LIN {X 0,Y 523.977,Z 285.218,A -85,B 0,C 180,E1 -4797.718,E2 -4797.718} C_VEL
LIN {X 0,Y 523.948,Z 285.216,A -85,B 0,C 180,E1 -4800.855,E2 -4800.855} C_VEL
LIN {X 0,Y 523.962,Z 285.215,A -85,B 0,C 180,E1 -4803.734,E2 -4803.734} C_VEL
LIN {X 0,Y 523.905,Z 285.226,A -85,B 0,C 180,E1 -4806.401,E2 -4806.401} C_VEL
LIN {X 0,Y 523.921,Z 285.217,A -85,B 0,C 180,E1 -4809.085,E2 -4809.085} C_VEL
LIN {X 0,Y 523.954,Z 285.219,A -85,B 0,C 180,E1 -4812.119,E2 -4812.119} C_VEL
LIN {X 0,Y 523.941,Z 285.215,A -85,B 0,C 180,E1 -4815.31,E2 -4815.31} C_VEL
LIN {X 0,Y 523.959,Z 285.219,A -85,B 0,C 180,E1 -4818.689,E2 -4818.689} C_VEL
LIN {X 0,Y 523.912,Z 285.219,A -85,B 0,C 180,E1 -4821.898,E2 -4821.898} C_VEL
LIN {X 0,Y 523.93,Z 285.222,A -85,B 0,C 180,E1 -4824.909,E2 -4824.909} C_VEL
LIN {X 0,Y 523.937,Z 285.215,A -85,B 0,C 180,E1 -4827.678,E2 -4827.678} C_VEL
LIN {X 0,Y 523.956,Z 285.221,A -85,B 0,C 180,E1 -4830.674,E2 -4830.674} C_VEL
LIN {X 0,Y 523.97,Z 285.211,A -85,B 0,C 180,E1 -4833.728,E2 -4833.728} C_VEL
LIN {X 0,Y 523.928,Z 285.217,A -85,B 0,C 180,E1 -4836.27,E2 -4836.27} C_VEL
LIN {X 0,Y 523.936,Z 285.222,A -85,B 0,C 180,E1 -4838.766,E2 -4838.766} C_VEL
LIN {X 0,Y 523.941,Z 285.222,A -85,B 0,C 180,E1 -4841.22,E2 -4841.22} C_VEL
LIN {X 0,Y 523.924,Z 285.219,A -85,B 0,C 180,E1 -4843.638,E2 -4843.638} C_VEL
LIN {X 0,Y 523.927,Z 285.216,A -85,B 0,C 180,E1 -4846.028,E2 -4846.028} C_VEL
LIN {X 0,Y 524.002,Z 285.207,A -85,B 0,C 180,E1 -4848.394,E2 -4848.394} C_VEL
LIN {X 0,Y 523.991,Z 285.215,A -85,B 0,C 180,E1 -4851.516,E2 -4851.516} C_VEL
LIN {X 0,Y 524.07,Z 285.199,A -85,B 0,C 180,E1 -4854.614,E2 -4854.614} C_VEL
LIN {X 0,Y 524.095,Z 285.201,A -85,B 0,C 180,E1 -4857.694,E2 -4857.694} C_VEL
LIN {X 0,Y 524.109,Z 285.194,A -85,B 0,C 180,E1 -4860.768,E2 -4860.768} C_VEL
LIN {X 0,Y 524.058,Z 285.203,A -85,B 0,C 180,E1 -4863.075,E2 -4863.075} C_VEL
LIN {X 0,Y 524.011,Z 285.208,A -85,B 0,C 180,E1 -4866.159,E2 -4866.159} C_VEL
LIN {X 0,Y 523.979,Z 285.213,A -85,B 0,C 180,E1 -4869.262,E2 -4869.262} C_VEL
LIN {X 0,Y 523.986,Z 285.219,A -85,B 0,C 180,E1 -4871.737,E2 -4871.737} C_VEL
LIN {X 0,Y 523.979,Z 285.21,A -85,B 0,C 180,E1 -4875.051,E2 -4875.051} C_VEL
LIN {X 0,Y 523.934,Z 285.225,A -85,B 0,C 180,E1 -4877.97,E2 -4877.97} C_VEL
LIN {X 0,Y 523.94,Z 285.218,A -85,B 0,C 180,E1 -4880.411,E2 -4880.411} C_VEL
LIN {X 0,Y 523.897,Z 285.22,A -85,B 0,C 180,E1 -4882.894,E2 -4882.894} C_VEL
LIN {X 0,Y 523.89,Z 285.222,A -85,B 0,C 180,E1 -4885.422,E2 -4885.422} C_VEL
LIN {X 0,Y 523.888,Z 285.229,A -85,B 0,C 180,E1 -4888.004,E2 -4888.004} C_VEL
LIN {X 0,Y 523.927,Z 285.218,A -85,B 0,C 180,E1 -4890.853,E2 -4890.853} C_VEL
LIN {X 0,Y 523.919,Z 285.219,A -85,B 0,C 180,E1 -4893.729,E2 -4893.729} C_VEL
LIN {X 0,Y 523.853,Z 285.235,A -85,B 0,C 180,E1 -4896.395,E2 -4896.395} C_VEL
LIN {X 0,Y 523.89,Z 285.222,A -85,B 0,C 180,E1 -4899.088,E2 -4899.088} C_VEL
LIN {X 0,Y 523.881,Z 285.226,A -85,B 0,C 180,E1 -4902.126,E2 -4902.126} C_VEL
LIN {X 0,Y 523.927,Z 285.217,A -85,B 0,C 180,E1 -4905.312,E2 -4905.312} C_VEL
LIN {X 0,Y 523.865,Z 285.229,A -85,B 0,C 180,E1 -4906.891,E2 -4906.891} C_VEL
LIN {X 0,Y 523.18,Z 285.312,A -85,B 0,C 180,E1 -4907.532,E2 -4907.532} C_VEL
LIN {X 0,Y 520.318,Z 285.675,A -85,B 0,C 180,E1 -4908.574,E2 -4908.574} C_VEL
LIN {X 0,Y 517.917,Z 285.971,A -85,B 0,C 180,E1 -4909.412,E2 -4909.412} C_VEL
LIN {X 0,Y 516.897,Z 286.095,A -85,B 0,C 180,E1 -4910.06,E2 -4910.06} C_VEL
LIN {X 0,Y 516.819,Z 286.105,A -85,B 0,C 180,E1 -4910.279,E2 -4910.279} C_VEL
LIN {X 0,Y 516.79,Z 286.108,A -85,B 0,C 180,E1 -4913.247,E2 -4913.247} C_VEL
LIN {X 0,Y 516.836,Z 286.101,A -85,B 0,C 180,E1 -4916.115,E2 -4916.115} C_VEL
LIN {X 0,Y 516.85,Z 286.107,A -85,B 0,C 180,E1 -4918.944,E2 -4918.944} C_VEL
LIN {X 0,Y 516.858,Z 286.097,A -85,B 0,C 180,E1 -4922.11,E2 -4922.11} C_VEL
LIN {X 0,Y 516.829,Z 286.11,A -85,B 0,C 180,E1 -4925.067,E2 -4925.067} C_VEL
LIN {X 0,Y 516.875,Z 286.097,A -85,B 0,C 180,E1 -4927.621,E2 -4927.621} C_VEL
LIN {X 0,Y 516.92,Z 286.089,A -85,B 0,C 180,E1 -4930.128,E2 -4930.128} C_VEL
LIN {X 0,Y 516.879,Z 286.101,A -85,B 0,C 180,E1 -4933.408,E2 -4933.408} C_VEL
LIN {X 0,Y 516.879,Z 286.096,A -85,B 0,C 180,E1 -4935.832,E2 -4935.832} C_VEL
LIN {X 0,Y 516.946,Z 286.09,A -85,B 0,C 180,E1 -4939.026,E2 -4939.026} C_VEL
LIN {X 0,Y 516.926,Z 286.089,A -85,B 0,C 180,E1 -4942.184,E2 -4942.184} C_VEL
LIN {X 0,Y 516.988,Z 286.081,A -85,B 0,C 180,E1 -4944.537,E2 -4944.537} C_VEL
LIN {X 0,Y 517.076,Z 286.078,A -85,B 0,C 180,E1 -4947.661,E2 -4947.661} C_VEL
LIN {X 0,Y 517.068,Z 286.075,A -85,B 0,C 180,E1 -4949.997,E2 -4949.997} C_VEL
LIN {X 0,Y 517.076,Z 286.071,A -85,B 0,C 180,E1 -4952.334,E2 -4952.334} C_VEL
LIN {X 0,Y 516.975,Z 286.087,A -85,B 0,C 180,E1 -4956.241,E2 -4956.241} C_VEL
LIN {X 0,Y 516.935,Z 286.093,A -85,B 0,C 180,E1 -4959.386,E2 -4959.386} C_VEL
LIN {X 0,Y 516.964,Z 286.096,A -85,B 0,C 180,E1 -4962.161,E2 -4962.161} C_VEL
LIN {X 0,Y 517.499,Z 292.038,A -85,B 0,C 180,E1 -4963.345,E2 -4963.345} C_VEL
LIN {X 0,Y 517.273,Z 306.74,A -85,B 0,C 180,E1 -4966.168,E2 -4966.168} C_VEL
LIN {X 0,Y 517.259,Z 309.78,A -85,B 0,C 180,E1 -4966.701,E2 -4966.701} C_VEL
LIN {X 0,Y 519.063,Z 319.454,A -85,B 0,C 180,E1 -4966.895,E2 -4966.895} C_VEL
LIN {X 0,Y 518.594,Z 416.572,A -85,B 0,C 180,E1 -4968.272,E2 -4968.272} C_VEL
LIN {X 0,Y 518.456,Z 429.396,A -85,B 0,C 180,E1 -4968.609,E2 -4968.609} C_VEL
LIN {X 0,Y 518.201,Z 441.954,A -85,B 0,C 180,E1 -4969.094,E2 -4969.094} C_VEL
LIN {X 0,Y 517.926,Z 453.888,A -85,B 0,C 180,E1 -4969.723,E2 -4969.723} C_VEL
LIN {X 0,Y 517.565,Z 465.513,A -85,B 0,C 180,E1 -4970.517,E2 -4970.517} C_VEL
LIN {X 0,Y 517.293,Z 475.939,A -85,B 0,C 180,E1 -4971.411,E2 -4971.411} C_VEL
LIN {X 0,Y 517.017,Z 485.499,A -85,B 0,C 180,E1 -4972.429,E2 -4972.429} C_VEL
LIN {X 0,Y 516.759,Z 494.699,A -85,B 0,C 180,E1 -4973.649,E2 -4973.649} C_VEL
LIN {X 0,Y 516.619,Z 500.444,A -85,B 0,C 180,E1 -4974.582,E2 -4974.582} C_VEL
LIN {X 0,Y 516.472,Z 506.637,A -85,B 0,C 180,E1 -4975.809,E2 -4975.809} C_VEL
LIN {X 0,Y 516.367,Z 511.787,A -85,B 0,C 180,E1 -4977.121,E2 -4977.121} C_VEL
LIN {X 0,Y 516.249,Z 515.595,A -85,B 0,C 180,E1 -4978.45,E2 -4978.45} C_VEL
LIN {X 0,Y 516.228,Z 517.529,A -85,B 0,C 180,E1 -4979.389,E2 -4979.389} C_VEL
LIN {X 0,Y 516.199,Z 518.78,A -85,B 0,C 180,E1 -4980.243,E2 -4980.243} C_VEL
LIN {X 0,Y 516.173,Z 519.558,A -85,B 0,C 180,E1 -4981.152,E2 -4981.152} C_VEL
LIN {X 0,Y 516.192,Z 519.773,A -85,B 0,C 180,E1 -4982.42,E2 -4982.42} C_VEL
LIN {X 0,Y 516.205,Z 518.701,A -85,B 0,C 180,E1 -4983.926,E2 -4983.926} C_VEL
LIN {X 0,Y 516.201,Z 516.554,A -85,B 0,C 180,E1 -4985.225,E2 -4985.225} C_VEL
LIN {X 0,Y 516.327,Z 513.062,A -85,B 0,C 180,E1 -4986.574,E2 -4986.574} C_VEL
LIN {X 0,Y 516.434,Z 508.387,A -85,B 0,C 180,E1 -4987.879,E2 -4987.879} C_VEL
LIN {X 0,Y 516.566,Z 502.458,A -85,B 0,C 180,E1 -4989.149,E2 -4989.149} C_VEL
LIN {X 0,Y 516.787,Z 495.044,A -85,B 0,C 180,E1 -4990.397,E2 -4990.397} C_VEL
LIN {X 0,Y 517.023,Z 485.936,A -85,B 0,C 180,E1 -4991.614,E2 -4991.614} C_VEL
LIN {X 0,Y 517.316,Z 476.332,A -85,B 0,C 180,E1 -4992.648,E2 -4992.648} C_VEL
LIN {X 0,Y 517.581,Z 466.186,A -85,B 0,C 180,E1 -4993.526,E2 -4993.526} C_VEL
LIN {X 0,Y 517.857,Z 455.616,A -85,B 0,C 180,E1 -4994.264,E2 -4994.264} C_VEL
LIN {X 0,Y 518.159,Z 443.921,A -85,B 0,C 180,E1 -4994.908,E2 -4994.908} C_VEL
LIN {X 0,Y 518.447,Z 431.069,A -85,B 0,C 180,E1 -4995.429,E2 -4995.429} C_VEL
LIN {X 0,Y 518.619,Z 417.781,A -85,B 0,C 180,E1 -4995.792,E2 -4995.792} C_VEL
LIN {X 0,Y 518.817,Z 379.999,A -85,B 0,C 180,E1 -4996.349,E2 -4996.349} C_VEL
LIN {X 0,Y 519.087,Z 319.542,A -85,B 0,C 180,E1 -4997.195,E2 -4997.195} C_VEL
LIN {X 0,Y 517.182,Z 309.105,A -85,B 0,C 180,E1 -4997.415,E2 -4997.415} C_VEL
LIN {X 0,Y 517.275,Z 293.741,A -85,B 0,C 180,E1 -5000.121,E2 -5000.121} C_VEL
LIN {X 0,Y 516.989,Z 286.453,A -85,B 0,C 180,E1 -5001.398,E2 -5001.398} C_VEL
LIN {X 0,Y 516.922,Z 286.097,A -85,B 0,C 180,E1 -5001.497,E2 -5001.497} C_VEL
LIN {X 0,Y 516.844,Z 286.105,A -85,B 0,C 180,E1 -5004.664,E2 -5004.664} C_VEL
LIN {X 0,Y 516.858,Z 286.099,A -85,B 0,C 180,E1 -5007.452,E2 -5007.452} C_VEL
LIN {X 0,Y 516.89,Z 286.099,A -85,B 0,C 180,E1 -5010.693,E2 -5010.693} C_VEL
LIN {X 0,Y 516.9,Z 286.097,A -85,B 0,C 180,E1 -5013.8,E2 -5013.8} C_VEL
LIN {X 0,Y 516.823,Z 286.109,A -85,B 0,C 180,E1 -5016.774,E2 -5016.774} C_VEL
LIN {X 0,Y 516.887,Z 286.096,A -85,B 0,C 180,E1 -5019.73,E2 -5019.73} C_VEL
LIN {X 0,Y 516.876,Z 286.105,A -85,B 0,C 180,E1 -5022.594,E2 -5022.594} C_VEL
LIN {X 0,Y 516.887,Z 286.098,A -85,B 0,C 180,E1 -5025.028,E2 -5025.028} C_VEL
LIN {X 0,Y 516.91,Z 286.095,A -85,B 0,C 180,E1 -5028.232,E2 -5028.232} C_VEL
LIN {X 0,Y 516.915,Z 286.091,A -85,B 0,C 180,E1 -5031.399,E2 -5031.399} C_VEL
LIN {X 0,Y 516.949,Z 286.086,A -85,B 0,C 180,E1 -5033.756,E2 -5033.756} C_VEL
LIN {X 0,Y 516.99,Z 286.089,A -85,B 0,C 180,E1 -5036.883,E2 -5036.883} C_VEL
LIN {X 0,Y 517.023,Z 286.074,A -85,B 0,C 180,E1 -5040,E2 -5040} C_VEL
LIN {X 0,Y 516.994,Z 286.085,A -85,B 0,C 180,E1 -5043.117,E2 -5043.117} C_VEL
LIN {X 0,Y 516.957,Z 286.086,A -85,B 0,C 180,E1 -5046.244,E2 -5046.244} C_VEL
LIN {X 0,Y 516.914,Z 286.095,A -85,B 0,C 180,E1 -5049.39,E2 -5049.39} C_VEL
LIN {X 0,Y 516.929,Z 286.086,A -85,B 0,C 180,E1 -5051.825,E2 -5051.825} C_VEL
LIN {X 0,Y 516.903,Z 286.099,A -85,B 0,C 180,E1 -5055.153,E2 -5055.153} C_VEL
LIN {X 0,Y 516.878,Z 286.094,A -85,B 0,C 180,E1 -5058.224,E2 -5058.224} C_VEL
LIN {X 0,Y 516.869,Z 286.095,A -85,B 0,C 180,E1 -5060.703,E2 -5060.703} C_VEL
LIN {X 0,Y 516.866,Z 286.104,A -85,B 0,C 180,E1 -5063.224,E2 -5063.224} C_VEL
LIN {X 0,Y 516.904,Z 286.091,A -85,B 0,C 180,E1 -5066.201,E2 -5066.201} C_VEL
LIN {X 0,Y 516.898,Z 286.098,A -85,B 0,C 180,E1 -5069.306,E2 -5069.306} C_VEL
LIN {X 0,Y 516.866,Z 286.096,A -85,B 0,C 180,E1 -5072.549,E2 -5072.549} C_VEL
LIN {X 0,Y 516.851,Z 286.105,A -85,B 0,C 180,E1 -5075.337,E2 -5075.337} C_VEL
LIN {X 0,Y 516.858,Z 286.101,A -85,B 0,C 180,E1 -5077.949,E2 -5077.949} C_VEL
LIN {X 0,Y 516.887,Z 286.095,A -85,B 0,C 180,E1 -5080.741,E2 -5080.741} C_VEL
LIN {X 0,Y 516.851,Z 286.107,A -85,B 0,C 180,E1 -5083.907,E2 -5083.907} C_VEL
LIN {X 0,Y 516.852,Z 286.104,A -85,B 0,C 180,E1 -5086.111,E2 -5086.111} C_VEL
LIN {X 0,Y 516.889,Z 286.098,A -85,B 0,C 180,E1 -5089.266,E2 -5089.266} C_VEL
LIN {X 0,Y 516.862,Z 286.104,A -85,B 0,C 180,E1 -5092.06,E2 -5092.06} C_VEL
LIN {X 0,Y 516.875,Z 286.098,A -85,B 0,C 180,E1 -5095.18,E2 -5095.18} C_VEL
LIN {X 0,Y 516.865,Z 286.107,A -85,B 0,C 180,E1 -5097.98,E2 -5097.98} C_VEL
LIN {X 0,Y 516.92,Z 286.094,A -85,B 0,C 180,E1 -5100.7,E2 -5100.7} C_VEL
LIN {X 0,Y 516.931,Z 286.097,A -85,B 0,C 180,E1 -5103.807,E2 -5103.807} C_VEL
LIN {X 0,Y 516.948,Z 286.248,A -85,B 0,C 180,E1 -5105.43,E2 -5105.43} C_VEL
LIN {X 0,Y 518.381,Z 294.852,A -85,B 0,C 180,E1 -5106.853,E2 -5106.853} C_VEL
LIN {X 0,Y 517.942,Z 314.961,A -85,B 0,C 180,E1 -5109.982,E2 -5109.982} C_VEL
LIN {X 0,Y 517.423,Z 334.741,A -85,B 0,C 180,E1 -5113.024,E2 -5113.024} C_VEL
LIN {X 0,Y 517.282,Z 345.377,A -85,B 0,C 180,E1 -5114.634,E2 -5114.634} C_VEL
LIN {X 0,Y 519.061,Z 357.7,A -85,B 0,C 180,E1 -5114.862,E2 -5114.862} C_VEL
LIN {X 0,Y 518.575,Z 454.458,A -85,B 0,C 180,E1 -5116.234,E2 -5116.234} C_VEL
LIN {X 0,Y 518.297,Z 468.259,A -85,B 0,C 180,E1 -5116.601,E2 -5116.601} C_VEL
LIN {X 0,Y 517.976,Z 481.158,A -85,B 0,C 180,E1 -5117.117,E2 -5117.117} C_VEL
LIN {X 0,Y 517.817,Z 492.708,A -85,B 0,C 180,E1 -5117.745,E2 -5117.745} C_VEL
LIN {X 0,Y 517.485,Z 504.303,A -85,B 0,C 180,E1 -5118.547,E2 -5118.547} C_VEL
LIN {X 0,Y 517.151,Z 514.547,A -85,B 0,C 180,E1 -5119.432,E2 -5119.432} C_VEL
LIN {X 0,Y 516.887,Z 523.76,A -85,B 0,C 180,E1 -5120.415,E2 -5120.415} C_VEL
LIN {X 0,Y 516.664,Z 532.738,A -85,B 0,C 180,E1 -5121.595,E2 -5121.595} C_VEL
LIN {X 0,Y 516.508,Z 539.965,A -85,B 0,C 180,E1 -5122.772,E2 -5122.772} C_VEL
LIN {X 0,Y 516.42,Z 546.546,A -85,B 0,C 180,E1 -5124.145,E2 -5124.145} C_VEL
LIN {X 0,Y 516.268,Z 550.897,A -85,B 0,C 180,E1 -5125.318,E2 -5125.318} C_VEL
LIN {X 0,Y 516.351,Z 553.206,A -85,B 0,C 180,E1 -5126.101,E2 -5126.101} C_VEL
LIN {X 0,Y 516.282,Z 555.072,A -85,B 0,C 180,E1 -5126.881,E2 -5126.881} C_VEL
LIN {X 0,Y 516.26,Z 556.472,A -85,B 0,C 180,E1 -5127.662,E2 -5127.662} C_VEL
LIN {X 0,Y 516.16,Z 558.08,A -85,B 0,C 180,E1 -5129.222,E2 -5129.222} C_VEL
LIN {X 0,Y 516.158,Z 558.297,A -85,B 0,C 180,E1 -5130.003,E2 -5130.003} C_VEL
LIN {X 0,Y 516.192,Z 557.473,A -85,B 0,C 180,E1 -5131.563,E2 -5131.563} C_VEL
LIN {X 0,Y 516.261,Z 556.479,A -85,B 0,C 180,E1 -5132.343,E2 -5132.343} C_VEL
LIN {X 0,Y 516.283,Z 555.079,A -85,B 0,C 180,E1 -5133.124,E2 -5133.124} C_VEL
LIN {X 0,Y 516.312,Z 552.136,A -85,B 0,C 180,E1 -5134.296,E2 -5134.296} C_VEL
LIN {X 0,Y 516.376,Z 548.152,A -85,B 0,C 180,E1 -5135.469,E2 -5135.469} C_VEL
LIN {X 0,Y 516.423,Z 542.925,A -85,B 0,C 180,E1 -5136.664,E2 -5136.664} C_VEL
LIN {X 0,Y 516.558,Z 536.56,A -85,B 0,C 180,E1 -5137.822,E2 -5137.822} C_VEL
LIN {X 0,Y 516.771,Z 528.505,A -85,B 0,C 180,E1 -5139,E2 -5139} C_VEL
LIN {X 0,Y 516.987,Z 520.294,A -85,B 0,C 180,E1 -5139.983,E2 -5139.983} C_VEL
LIN {X 0,Y 517.273,Z 510.282,A -85,B 0,C 180,E1 -5140.967,E2 -5140.967} C_VEL
LIN {X 0,Y 517.626,Z 500.396,A -85,B 0,C 180,E1 -5141.753,E2 -5141.753} C_VEL
LIN {X 0,Y 517.852,Z 489.209,A -85,B 0,C 180,E1 -5142.468,E2 -5142.468} C_VEL
LIN {X 0,Y 518.152,Z 476.709,A -85,B 0,C 180,E1 -5143.083,E2 -5143.083} C_VEL
LIN {X 0,Y 518.381,Z 464.379,A -85,B 0,C 180,E1 -5143.527,E2 -5143.527} C_VEL
LIN {X 0,Y 518.589,Z 451.7,A -85,B 0,C 180,E1 -5143.821,E2 -5143.821} C_VEL
LIN {X 0,Y 519.006,Z 357.028,A -85,B 0,C 180,E1 -5145.151,E2 -5145.151} C_VEL
LIN {X 0,Y 517.295,Z 345.507,A -85,B 0,C 180,E1 -5145.367,E2 -5145.367} C_VEL
LIN {X 0,Y 517.761,Z 324.652,A -85,B 0,C 180,E1 -5148.603,E2 -5148.603} C_VEL
LIN {X 0,Y 518.218,Z 306.327,A -85,B 0,C 180,E1 -5151.481,E2 -5151.481} C_VEL
LIN {X 0,Y 518.477,Z 294.562,A -85,B 0,C 180,E1 -5153.36,E2 -5153.36} C_VEL
LIN {X 0,Y 516.925,Z 286.095,A -85,B 0,C 180,E1 -5154.821,E2 -5154.821} C_VEL
LIN {X 0,Y 516.927,Z 286.095,A -85,B 0,C 180,E1 -5157.533,E2 -5157.533} C_VEL
LIN {X 0,Y 516.896,Z 286.102,A -85,B 0,C 180,E1 -5160.204,E2 -5160.204} C_VEL
LIN {X 0,Y 516.898,Z 286.092,A -85,B 0,C 180,E1 -5162.947,E2 -5162.947} C_VEL
LIN {X 0,Y 516.873,Z 286.099,A -85,B 0,C 180,E1 -5165.78,E2 -5165.78} C_VEL
LIN {X 0,Y 516.881,Z 286.097,A -85,B 0,C 180,E1 -5168.716,E2 -5168.716} C_VEL
LIN {X 0,Y 516.914,Z 286.092,A -85,B 0,C 180,E1 -5171.775,E2 -5171.775} C_VEL
LIN {X 0,Y 516.894,Z 286.094,A -85,B 0,C 180,E1 -5175.007,E2 -5175.007} C_VEL
LIN {X 0,Y 516.915,Z 286.098,A -85,B 0,C 180,E1 -5178.398,E2 -5178.398} C_VEL
LIN {X 0,Y 516.878,Z 286.095,A -85,B 0,C 180,E1 -5181.284,E2 -5181.284} C_VEL
LIN {X 0,Y 516.883,Z 286.097,A -85,B 0,C 180,E1 -5184.22,E2 -5184.22} C_VEL
LIN {X 0,Y 516.892,Z 286.097,A -85,B 0,C 180,E1 -5187.053,E2 -5187.053} C_VEL
LIN {X 0,Y 516.895,Z 286.092,A -85,B 0,C 180,E1 -5189.796,E2 -5189.796} C_VEL
LIN {X 0,Y 516.922,Z 286.093,A -85,B 0,C 180,E1 -5192.467,E2 -5192.467} C_VEL
LIN {X 0,Y 516.904,Z 286.098,A -85,B 0,C 180,E1 -5195.071,E2 -5195.071} C_VEL
LIN {X 0,Y 516.876,Z 286.097,A -85,B 0,C 180,E1 -5198.462,E2 -5198.462} C_VEL
LIN {X 0,Y 516.893,Z 286.101,A -85,B 0,C 180,E1 -5200.954,E2 -5200.954} C_VEL
LIN {X 0,Y 516.902,Z 286.096,A -85,B 0,C 180,E1 -5203.41,E2 -5203.41} C_VEL
LIN {X 0,Y 516.883,Z 286.095,A -85,B 0,C 180,E1 -5205.833,E2 -5205.833} C_VEL
LIN {X 0,Y 516.955,Z 286.085,A -85,B 0,C 180,E1 -5208.233,E2 -5208.233} C_VEL
LIN {X 0,Y 516.956,Z 286.093,A -85,B 0,C 180,E1 -5211.399,E2 -5211.399} C_VEL
LIN {X 0,Y 516.988,Z 286.084,A -85,B 0,C 180,E1 -5213.757,E2 -5213.757} C_VEL
LIN {X 0,Y 517.002,Z 286.081,A -85,B 0,C 180,E1 -5216.883,E2 -5216.883} C_VEL
LIN {X 0,Y 517.065,Z 286.074,A -85,B 0,C 180,E1 -5220,E2 -5220} C_VEL
LIN {X 0,Y 517,Z 286.082,A -85,B 0,C 180,E1 -5223.117,E2 -5223.117} C_VEL
LIN {X 0,Y 516.974,Z 286.084,A -85,B 0,C 180,E1 -5226.244,E2 -5226.244} C_VEL
LIN {X 0,Y 516.934,Z 286.092,A -85,B 0,C 180,E1 -5229.39,E2 -5229.39} C_VEL
LIN {X 0,Y 516.941,Z 286.096,A -85,B 0,C 180,E1 -5231.807,E2 -5231.807} C_VEL
LIN {X 0,Y 516.931,Z 286.089,A -85,B 0,C 180,E1 -5235.145,E2 -5235.145} C_VEL
LIN {X 0,Y 516.902,Z 286.096,A -85,B 0,C 180,E1 -5238.223,E2 -5238.223} C_VEL
LIN {X 0,Y 516.89,Z 286.094,A -85,B 0,C 180,E1 -5240.703,E2 -5240.703} C_VEL
LIN {X 0,Y 516.847,Z 286.099,A -85,B 0,C 180,E1 -5243.225,E2 -5243.225} C_VEL
LIN {X 0,Y 516.87,Z 286.104,A -85,B 0,C 180,E1 -5246.182,E2 -5246.182} C_VEL
LIN {X 0,Y 516.878,Z 286.096,A -85,B 0,C 180,E1 -5249.519,E2 -5249.519} C_VEL
LIN {X 0,Y 516.887,Z 286.099,A -85,B 0,C 180,E1 -5252.543,E2 -5252.543} C_VEL
LIN {X 0,Y 516.843,Z 286.099,A -85,B 0,C 180,E1 -5255.327,E2 -5255.327} C_VEL
LIN {X 0,Y 516.857,Z 286.102,A -85,B 0,C 180,E1 -5258.718,E2 -5258.718} C_VEL
LIN {X 0,Y 516.831,Z 286.101,A -85,B 0,C 180,E1 -5261.784,E2 -5261.784} C_VEL
LIN {X 0,Y 516.895,Z 286.095,A -85,B 0,C 180,E1 -5265.007,E2 -5265.007} C_VEL
LIN {X 0,Y 516.827,Z 286.107,A -85,B 0,C 180,E1 -5268.41,E2 -5268.41} C_VEL
LIN {X 0,Y 516.819,Z 286.105,A -85,B 0,C 180,E1 -5270.279,E2 -5270.279} C_VEL
LIN {X 0,Y 516.165,Z 286.191,A -85,B 0,C 180,E1 -5270.93,E2 -5270.93} C_VEL
LIN {X 0,Y 513.309,Z 286.543,A -85,B 0,C 180,E1 -5271.985,E2 -5271.985} C_VEL
LIN {X 0,Y 510.883,Z 286.85,A -85,B 0,C 180,E1 -5272.835,E2 -5272.835} C_VEL
LIN {X 0,Y 509.834,Z 286.973,A -85,B 0,C 180,E1 -5273.492,E2 -5273.492} C_VEL
LIN {X 0,Y 509.746,Z 286.983,A -85,B 0,C 180,E1 -5273.715,E2 -5273.715} C_VEL
LIN {X 0,Y 509.805,Z 286.98,A -85,B 0,C 180,E1 -5276.535,E2 -5276.535} C_VEL
LIN {X 0,Y 509.803,Z 286.979,A -85,B 0,C 180,E1 -5279.331,E2 -5279.331} C_VEL
LIN {X 0,Y 509.825,Z 286.973,A -85,B 0,C 180,E1 -5282.05,E2 -5282.05} C_VEL
LIN {X 0,Y 509.782,Z 286.983,A -85,B 0,C 180,E1 -5284.698,E2 -5284.698} C_VEL
LIN {X 0,Y 509.83,Z 286.977,A -85,B 0,C 180,E1 -5287.458,E2 -5287.458} C_VEL
LIN {X 0,Y 509.911,Z 286.963,A -85,B 0,C 180,E1 -5289.843,E2 -5289.843} C_VEL
LIN {X 0,Y 509.851,Z 286.979,A -85,B 0,C 180,E1 -5293.172,E2 -5293.172} C_VEL
LIN {X 0,Y 509.852,Z 286.974,A -85,B 0,C 180,E1 -5295.632,E2 -5295.632} C_VEL
LIN {X 0,Y 509.911,Z 286.965,A -85,B 0,C 180,E1 -5298.873,E2 -5298.873} C_VEL
LIN {X 0,Y 509.879,Z 286.968,A -85,B 0,C 180,E1 -5302.075,E2 -5302.075} C_VEL
LIN {X 0,Y 509.943,Z 286.958,A -85,B 0,C 180,E1 -5304.462,E2 -5304.462} C_VEL
LIN {X 0,Y 510.045,Z 286.955,A -85,B 0,C 180,E1 -5307.628,E2 -5307.628} C_VEL
LIN {X 0,Y 510.037,Z 286.951,A -85,B 0,C 180,E1 -5309.997,E2 -5309.997} C_VEL
LIN {X 0,Y 510.044,Z 286.947,A -85,B 0,C 180,E1 -5312.366,E2 -5312.366} C_VEL
LIN {X 0,Y 509.942,Z 286.965,A -85,B 0,C 180,E1 -5315.533,E2 -5315.533} C_VEL
LIN {X 0,Y 509.9,Z 286.966,A -85,B 0,C 180,E1 -5318.717,E2 -5318.717} C_VEL
LIN {X 0,Y 509.926,Z 287.092,A -85,B 0,C 180,E1 -5322.054,E2 -5322.054} C_VEL
LIN {X 0,Y 510.522,Z 293.451,A -85,B 0,C 180,E1 -5323.328,E2 -5323.328} C_VEL
LIN {X 0,Y 510.276,Z 308.215,A -85,B 0,C 180,E1 -5326.191,E2 -5326.191} C_VEL
LIN {X 0,Y 510.26,Z 309.688,A -85,B 0,C 180,E1 -5326.474,E2 -5326.474} C_VEL
LIN {X 0,Y 512.299,Z 321.362,A -85,B 0,C 180,E1 -5326.714,E2 -5326.714} C_VEL
LIN {X 0,Y 511.706,Z 416.31,A -85,B 0,C 180,E1 -5328.074,E2 -5328.074} C_VEL
LIN {X 0,Y 511.572,Z 429.601,A -85,B 0,C 180,E1 -5328.425,E2 -5328.425} C_VEL
LIN {X 0,Y 511.309,Z 441.708,A -85,B 0,C 180,E1 -5328.897,E2 -5328.897} C_VEL
LIN {X 0,Y 510.982,Z 452.9,A -85,B 0,C 180,E1 -5329.479,E2 -5329.479} C_VEL
LIN {X 0,Y 510.663,Z 464.377,A -85,B 0,C 180,E1 -5330.253,E2 -5330.253} C_VEL
LIN {X 0,Y 510.344,Z 475.349,A -85,B 0,C 180,E1 -5331.188,E2 -5331.188} C_VEL
LIN {X 0,Y 510.039,Z 483.565,A -85,B 0,C 180,E1 -5332.043,E2 -5332.043} C_VEL
LIN {X 0,Y 509.8,Z 492.2,A -85,B 0,C 180,E1 -5333.13,E2 -5333.13} C_VEL
LIN {X 0,Y 509.632,Z 499.226,A -85,B 0,C 180,E1 -5334.217,E2 -5334.217} C_VEL
LIN {X 0,Y 509.431,Z 506.034,A -85,B 0,C 180,E1 -5335.534,E2 -5335.534} C_VEL
LIN {X 0,Y 509.327,Z 510.574,A -85,B 0,C 180,E1 -5336.639,E2 -5336.639} C_VEL
LIN {X 0,Y 509.195,Z 514.796,A -85,B 0,C 180,E1 -5337.982,E2 -5337.982} C_VEL
LIN {X 0,Y 509.138,Z 516.934,A -85,B 0,C 180,E1 -5338.885,E2 -5338.885} C_VEL
LIN {X 0,Y 509.109,Z 518.476,A -85,B 0,C 180,E1 -5339.794,E2 -5339.794} C_VEL
LIN {X 0,Y 509.096,Z 519.821,A -85,B 0,C 180,E1 -5341.14,E2 -5341.14} C_VEL
LIN {X 0,Y 509.092,Z 519.996,A -85,B 0,C 180,E1 -5342.637,E2 -5342.637} C_VEL
LIN {X 0,Y 509.105,Z 518.798,A -85,B 0,C 180,E1 -5344.077,E2 -5344.077} C_VEL
LIN {X 0,Y 509.161,Z 516.36,A -85,B 0,C 180,E1 -5345.473,E2 -5345.473} C_VEL
LIN {X 0,Y 509.277,Z 512.722,A -85,B 0,C 180,E1 -5346.832,E2 -5346.832} C_VEL
LIN {X 0,Y 509.395,Z 507.892,A -85,B 0,C 180,E1 -5348.148,E2 -5348.148} C_VEL
LIN {X 0,Y 509.547,Z 501.754,A -85,B 0,C 180,E1 -5349.431,E2 -5349.431} C_VEL
LIN {X 0,Y 509.777,Z 494.111,A -85,B 0,C 180,E1 -5350.689,E2 -5350.689} C_VEL
LIN {X 0,Y 510.022,Z 485.574,A -85,B 0,C 180,E1 -5351.823,E2 -5351.823} C_VEL
LIN {X 0,Y 510.33,Z 476.328,A -85,B 0,C 180,E1 -5352.818,E2 -5352.818} C_VEL
LIN {X 0,Y 510.67,Z 465.619,A -85,B 0,C 180,E1 -5353.746,E2 -5353.746} C_VEL
LIN {X 0,Y 510.945,Z 455.444,A -85,B 0,C 180,E1 -5354.458,E2 -5354.458} C_VEL
LIN {X 0,Y 511.265,Z 443.24,A -85,B 0,C 180,E1 -5355.129,E2 -5355.129} C_VEL
LIN {X 0,Y 511.547,Z 430.586,A -85,B 0,C 180,E1 -5355.636,E2 -5355.636} C_VEL
LIN {X 0,Y 511.737,Z 417.569,A -85,B 0,C 180,E1 -5355.989,E2 -5355.989} C_VEL
LIN {X 0,Y 512.162,Z 351.038,A -85,B 0,C 180,E1 -5356.955,E2 -5356.955} C_VEL
LIN {X 0,Y 512.138,Z 320.023,A -85,B 0,C 180,E1 -5357.403,E2 -5357.403} C_VEL
LIN {X 0,Y 510.205,Z 309.336,A -85,B 0,C 180,E1 -5357.627,E2 -5357.627} C_VEL
LIN {X 0,Y 510.322,Z 291.928,A -85,B 0,C 180,E1 -5360.691,E2 -5360.691} C_VEL
LIN {X 0,Y 509.87,Z 286.976,A -85,B 0,C 180,E1 -5361.601,E2 -5361.601} C_VEL
LIN {X 0,Y 509.807,Z 286.982,A -85,B 0,C 180,E1 -5364.62,E2 -5364.62} C_VEL
LIN {X 0,Y 509.824,Z 286.976,A -85,B 0,C 180,E1 -5367.478,E2 -5367.478} C_VEL
LIN {X 0,Y 509.837,Z 286.981,A -85,B 0,C 180,E1 -5370.266,E2 -5370.266} C_VEL
LIN {X 0,Y 509.842,Z 286.977,A -85,B 0,C 180,E1 -5372.942,E2 -5372.942} C_VEL
LIN {X 0,Y 509.824,Z 286.978,A -85,B 0,C 180,E1 -5375.572,E2 -5375.572} C_VEL
LIN {X 0,Y 509.799,Z 286.981,A -85,B 0,C 180,E1 -5378.996,E2 -5378.996} C_VEL
LIN {X 0,Y 509.836,Z 286.975,A -85,B 0,C 180,E1 -5381.997,E2 -5381.997} C_VEL
LIN {X 0,Y 509.857,Z 286.976,A -85,B 0,C 180,E1 -5384.817,E2 -5384.817} C_VEL
LIN {X 0,Y 509.85,Z 286.973,A -85,B 0,C 180,E1 -5388.12,E2 -5388.12} C_VEL
LIN {X 0,Y 509.862,Z 286.971,A -85,B 0,C 180,E1 -5391.279,E2 -5391.279} C_VEL
LIN {X 0,Y 509.9,Z 286.964,A -85,B 0,C 180,E1 -5393.669,E2 -5393.669} C_VEL
LIN {X 0,Y 509.931,Z 286.968,A -85,B 0,C 180,E1 -5396.84,E2 -5396.84} C_VEL
LIN {X 0,Y 509.994,Z 286.95,A -85,B 0,C 180,E1 -5400,E2 -5400} C_VEL
LIN {X 0,Y 509.934,Z 286.963,A -85,B 0,C 180,E1 -5403.16,E2 -5403.16} C_VEL
LIN {X 0,Y 509.925,Z 286.962,A -85,B 0,C 180,E1 -5406.33,E2 -5406.33} C_VEL
LIN {X 0,Y 509.898,Z 286.967,A -85,B 0,C 180,E1 -5408.721,E2 -5408.721} C_VEL
LIN {X 0,Y 509.897,Z 286.962,A -85,B 0,C 180,E1 -5411.932,E2 -5411.932} C_VEL
LIN {X 0,Y 509.849,Z 286.976,A -85,B 0,C 180,E1 -5415.247,E2 -5415.247} C_VEL
LIN {X 0,Y 509.839,Z 286.972,A -85,B 0,C 180,E1 -5418.004,E2 -5418.004} C_VEL
LIN {X 0,Y 509.814,Z 286.977,A -85,B 0,C 180,E1 -5421.003,E2 -5421.003} C_VEL
LIN {X 0,Y 509.823,Z 286.976,A -85,B 0,C 180,E1 -5423.564,E2 -5423.564} C_VEL
LIN {X 0,Y 509.872,Z 286.967,A -85,B 0,C 180,E1 -5426.383,E2 -5426.383} C_VEL
LIN {X 0,Y 509.846,Z 286.97,A -85,B 0,C 180,E1 -5428.846,E2 -5428.846} C_VEL
LIN {X 0,Y 509.787,Z 286.984,A -85,B 0,C 180,E1 -5431.593,E2 -5431.593} C_VEL
LIN {X 0,Y 509.815,Z 286.975,A -85,B 0,C 180,E1 -5434.416,E2 -5434.416} C_VEL
LIN {X 0,Y 509.794,Z 286.984,A -85,B 0,C 180,E1 -5437.343,E2 -5437.343} C_VEL
LIN {X 0,Y 509.854,Z 286.971,A -85,B 0,C 180,E1 -5440.381,E2 -5440.381} C_VEL
LIN {X 0,Y 509.808,Z 286.979,A -85,B 0,C 180,E1 -5443.068,E2 -5443.068} C_VEL
LIN {X 0,Y 509.8,Z 286.986,A -85,B 0,C 180,E1 -5445.796,E2 -5445.796} C_VEL
LIN {X 0,Y 509.844,Z 286.973,A -85,B 0,C 180,E1 -5448.58,E2 -5448.58} C_VEL
LIN {X 0,Y 509.833,Z 286.981,A -85,B 0,C 180,E1 -5451.789,E2 -5451.789} C_VEL
LIN {X 0,Y 509.825,Z 286.976,A -85,B 0,C 180,E1 -5454.628,E2 -5454.628} C_VEL
LIN {X 0,Y 509.847,Z 286.977,A -85,B 0,C 180,E1 -5457.485,E2 -5457.485} C_VEL
LIN {X 0,Y 509.865,Z 286.978,A -85,B 0,C 180,E1 -5460.273,E2 -5460.273} C_VEL
LIN {X 0,Y 509.873,Z 286.971,A -85,B 0,C 180,E1 -5462.949,E2 -5462.949} C_VEL
LIN {X 0,Y 509.92,Z 287.17,A -85,B 0,C 180,E1 -5465.277,E2 -5465.277} C_VEL
LIN {X 0,Y 511.437,Z 296.522,A -85,B 0,C 180,E1 -5466.84,E2 -5466.84} C_VEL
LIN {X 0,Y 510.948,Z 315.877,A -85,B 0,C 180,E1 -5469.891,E2 -5469.891} C_VEL
LIN {X 0,Y 510.438,Z 334.452,A -85,B 0,C 180,E1 -5472.785,E2 -5472.785} C_VEL
LIN {X 0,Y 510.23,Z 345.001,A -85,B 0,C 180,E1 -5474.415,E2 -5474.415} C_VEL
LIN {X 0,Y 512.225,Z 358.623,A -85,B 0,C 180,E1 -5474.673,E2 -5474.673} C_VEL
LIN {X 0,Y 511.684,Z 454.057,A -85,B 0,C 180,E1 -5476.045,E2 -5476.045} C_VEL
LIN {X 0,Y 511.396,Z 467.897,A -85,B 0,C 180,E1 -5476.417,E2 -5476.417} C_VEL
LIN {X 0,Y 511.045,Z 480.825,A -85,B 0,C 180,E1 -5476.939,E2 -5476.939} C_VEL
LIN {X 0,Y 510.838,Z 492.485,A -85,B 0,C 180,E1 -5477.582,E2 -5477.582} C_VEL
LIN {X 0,Y 510.505,Z 503.991,A -85,B 0,C 180,E1 -5478.388,E2 -5478.388} C_VEL
LIN {X 0,Y 510.153,Z 514.246,A -85,B 0,C 180,E1 -5479.285,E2 -5479.285} C_VEL
LIN {X 0,Y 509.856,Z 523.465,A -85,B 0,C 180,E1 -5480.282,E2 -5480.282} C_VEL
LIN {X 0,Y 509.62,Z 532.45,A -85,B 0,C 180,E1 -5481.478,E2 -5481.478} C_VEL
LIN {X 0,Y 509.429,Z 539.682,A -85,B 0,C 180,E1 -5482.672,E2 -5482.672} C_VEL
LIN {X 0,Y 509.307,Z 544.562,A -85,B 0,C 180,E1 -5483.665,E2 -5483.665} C_VEL
LIN {X 0,Y 509.242,Z 549.307,A -85,B 0,C 180,E1 -5484.856,E2 -5484.856} C_VEL
LIN {X 0,Y 509.245,Z 552.934,A -85,B 0,C 180,E1 -5486.046,E2 -5486.046} C_VEL
LIN {X 0,Y 509.2,Z 554.803,A -85,B 0,C 180,E1 -5486.838,E2 -5486.838} C_VEL
LIN {X 0,Y 509.189,Z 556.205,A -85,B 0,C 180,E1 -5487.63,E2 -5487.63} C_VEL
LIN {X 0,Y 509.073,Z 557.815,A -85,B 0,C 180,E1 -5489.212,E2 -5489.212} C_VEL
LIN {X 0,Y 509.069,Z 558.033,A -85,B 0,C 180,E1 -5490.003,E2 -5490.003} C_VEL
LIN {X 0,Y 509.112,Z 557.21,A -85,B 0,C 180,E1 -5491.585,E2 -5491.585} C_VEL
LIN {X 0,Y 509.19,Z 556.216,A -85,B 0,C 180,E1 -5492.376,E2 -5492.376} C_VEL
LIN {X 0,Y 509.201,Z 554.816,A -85,B 0,C 180,E1 -5493.167,E2 -5493.167} C_VEL
LIN {X 0,Y 509.204,Z 551.871,A -85,B 0,C 180,E1 -5494.356,E2 -5494.356} C_VEL
LIN {X 0,Y 509.294,Z 547.885,A -85,B 0,C 180,E1 -5495.545,E2 -5495.545} C_VEL
LIN {X 0,Y 509.402,Z 541.852,A -85,B 0,C 180,E1 -5496.916,E2 -5496.916} C_VEL
LIN {X 0,Y 509.545,Z 535.048,A -85,B 0,C 180,E1 -5498.129,E2 -5498.129} C_VEL
LIN {X 0,Y 509.75,Z 526.733,A -85,B 0,C 180,E1 -5499.325,E2 -5499.325} C_VEL
LIN {X 0,Y 509.987,Z 518.202,A -85,B 0,C 180,E1 -5500.322,E2 -5500.322} C_VEL
LIN {X 0,Y 510.389,Z 507.667,A -85,B 0,C 180,E1 -5501.318,E2 -5501.318} C_VEL
LIN {X 0,Y 510.67,Z 497.337,A -85,B 0,C 180,E1 -5502.11,E2 -5502.11} C_VEL
LIN {X 0,Y 510.998,Z 485.797,A -85,B 0,C 180,E1 -5502.815,E2 -5502.815} C_VEL
LIN {X 0,Y 511.227,Z 473.995,A -85,B 0,C 180,E1 -5503.365,E2 -5503.365} C_VEL
LIN {X 0,Y 511.556,Z 460.396,A -85,B 0,C 180,E1 -5503.812,E2 -5503.812} C_VEL
LIN {X 0,Y 511.755,Z 446.638,A -85,B 0,C 180,E1 -5504.085,E2 -5504.085} C_VEL
LIN {X 0,Y 512.139,Z 357.556,A -85,B 0,C 180,E1 -5505.348,E2 -5505.348} C_VEL
LIN {X 0,Y 510.26,Z 345.159,A -85,B 0,C 180,E1 -5505.599,E2 -5505.599} C_VEL
LIN {X 0,Y 510.789,Z 324.393,A -85,B 0,C 180,E1 -5508.866,E2 -5508.866} C_VEL
LIN {X 0,Y 511.308,Z 306.102,A -85,B 0,C 180,E1 -5511.786,E2 -5511.786} C_VEL
LIN {X 0,Y 511.501,Z 295.644,A -85,B 0,C 180,E1 -5513.483,E2 -5513.483} C_VEL
LIN {X 0,Y 509.898,Z 286.971,A -85,B 0,C 180,E1 -5515.007,E2 -5515.007} C_VEL
LIN {X 0,Y 509.888,Z 286.975,A -85,B 0,C 180,E1 -5517.947,E2 -5517.947} C_VEL
LIN {X 0,Y 509.849,Z 286.974,A -85,B 0,C 180,E1 -5520.666,E2 -5520.666} C_VEL
LIN {X 0,Y 509.862,Z 286.969,A -85,B 0,C 180,E1 -5523.461,E2 -5523.461} C_VEL
LIN {X 0,Y 509.827,Z 286.98,A -85,B 0,C 180,E1 -5526.353,E2 -5526.353} C_VEL
LIN {X 0,Y 509.847,Z 286.97,A -85,B 0,C 180,E1 -5529.352,E2 -5529.352} C_VEL
LIN {X 0,Y 509.834,Z 286.98,A -85,B 0,C 180,E1 -5532.49,E2 -5532.49} C_VEL
LIN {X 0,Y 509.838,Z 286.971,A -85,B 0,C 180,E1 -5535.33,E2 -5535.33} C_VEL
LIN {X 0,Y 509.857,Z 286.978,A -85,B 0,C 180,E1 -5538.574,E2 -5538.574} C_VEL
LIN {X 0,Y 509.848,Z 286.971,A -85,B 0,C 180,E1 -5541.786,E2 -5541.786} C_VEL
LIN {X 0,Y 509.838,Z 286.981,A -85,B 0,C 180,E1 -5544.622,E2 -5544.622} C_VEL
LIN {X 0,Y 509.86,Z 286.969,A -85,B 0,C 180,E1 -5547.481,E2 -5547.481} C_VEL
LIN {X 0,Y 509.855,Z 286.972,A -85,B 0,C 180,E1 -5550.273,E2 -5550.273} C_VEL
LIN {X 0,Y 509.88,Z 286.974,A -85,B 0,C 180,E1 -5552.944,E2 -5552.944} C_VEL
LIN {X 0,Y 509.862,Z 286.97,A -85,B 0,C 180,E1 -5555.574,E2 -5555.574} C_VEL
LIN {X 0,Y 509.841,Z 286.981,A -85,B 0,C 180,E1 -5558.998,E2 -5558.998} C_VEL
LIN {X 0,Y 509.872,Z 286.967,A -85,B 0,C 180,E1 -5562.001,E2 -5562.001} C_VEL
LIN {X 0,Y 509.901,Z 286.968,A -85,B 0,C 180,E1 -5564.818,E2 -5564.818} C_VEL
LIN {X 0,Y 509.89,Z 286.965,A -85,B 0,C 180,E1 -5568.124,E2 -5568.124} C_VEL
LIN {X 0,Y 509.903,Z 286.973,A -85,B 0,C 180,E1 -5571.28,E2 -5571.28} C_VEL
LIN {X 0,Y 509.94,Z 286.963,A -85,B 0,C 180,E1 -5573.67,E2 -5573.67} C_VEL
LIN {X 0,Y 509.944,Z 286.96,A -85,B 0,C 180,E1 -5576.84,E2 -5576.84} C_VEL
LIN {X 0,Y 510.053,Z 286.95,A -85,B 0,C 180,E1 -5579.211,E2 -5579.211} C_VEL
LIN {X 0,Y 510.037,Z 286.947,A -85,B 0,C 180,E1 -5582.369,E2 -5582.369} C_VEL
LIN {X 0,Y 509.959,Z 286.965,A -85,B 0,C 180,E1 -5585.536,E2 -5585.536} C_VEL
LIN {X 0,Y 509.894,Z 286.965,A -85,B 0,C 180,E1 -5588.721,E2 -5588.721} C_VEL
LIN {X 0,Y 509.894,Z 286.972,A -85,B 0,C 180,E1 -5591.932,E2 -5591.932} C_VEL
LIN {X 0,Y 509.885,Z 286.967,A -85,B 0,C 180,E1 -5595.242,E2 -5595.242} C_VEL
LIN {X 0,Y 509.846,Z 286.972,A -85,B 0,C 180,E1 -5598.484,E2 -5598.484} C_VEL
LIN {X 0,Y 509.833,Z 286.972,A -85,B 0,C 180,E1 -5601.003,E2 -5601.003} C_VEL
LIN {X 0,Y 509.809,Z 286.978,A -85,B 0,C 180,E1 -5603.565,E2 -5603.565} C_VEL
LIN {X 0,Y 509.806,Z 286.981,A -85,B 0,C 180,E1 -5606.356,E2 -5606.356} C_VEL
LIN {X 0,Y 509.825,Z 286.974,A -85,B 0,C 180,E1 -5608.848,E2 -5608.848} C_VEL
LIN {X 0,Y 509.811,Z 286.976,A -85,B 0,C 180,E1 -5611.591,E2 -5611.591} C_VEL
LIN {X 0,Y 509.827,Z 286.981,A -85,B 0,C 180,E1 -5614.416,E2 -5614.416} C_VEL
LIN {X 0,Y 509.771,Z 286.98,A -85,B 0,C 180,E1 -5617.345,E2 -5617.345} C_VEL
LIN {X 0,Y 509.787,Z 286.987,A -85,B 0,C 180,E1 -5620.387,E2 -5620.387} C_VEL
LIN {X 0,Y 509.788,Z 286.978,A -85,B 0,C 180,E1 -5623.575,E2 -5623.575} C_VEL
LIN {X 0,Y 509.789,Z 286.985,A -85,B 0,C 180,E1 -5626.425,E2 -5626.425} C_VEL
LIN {X 0,Y 509.785,Z 286.978,A -85,B 0,C 180,E1 -5629.613,E2 -5629.613} C_VEL
LIN {X 0,Y 509.756,Z 286.99,A -85,B 0,C 180,E1 -5632.654,E2 -5632.654} C_VEL
LIN {X 0,Y 509.746,Z 286.983,A -85,B 0,C 180,E1 -5633.715,E2 -5633.715} C_VEL
LIN {X 0,Y 509.08,Z 287.071,A -85,B 0,C 180,E1 -5634.374,E2 -5634.374} C_VEL
LIN {X 0,Y 506.259,Z 287.425,A -85,B 0,C 180,E1 -5635.446,E2 -5635.446} C_VEL
LIN {X 0,Y 503.872,Z 287.725,A -85,B 0,C 180,E1 -5636.31,E2 -5636.31} C_VEL
LIN {X 0,Y 502.838,Z 287.851,A -85,B 0,C 180,E1 -5636.977,E2 -5636.977} C_VEL
LIN {X 0,Y 502.749,Z 287.859,A -85,B 0,C 180,E1 -5637.202,E2 -5637.202} C_VEL
LIN {X 0,Y 502.745,Z 287.855,A -85,B 0,C 180,E1 -5640.079,E2 -5640.079} C_VEL
LIN {X 0,Y 502.771,Z 287.855,A -85,B 0,C 180,E1 -5642.529,E2 -5642.529} C_VEL
LIN {X 0,Y 502.765,Z 287.858,A -85,B 0,C 180,E1 -5645.315,E2 -5645.315} C_VEL
LIN {X 0,Y 502.784,Z 287.851,A -85,B 0,C 180,E1 -5647.825,E2 -5647.825} C_VEL
LIN {X 0,Y 502.811,Z 287.847,A -85,B 0,C 180,E1 -5650.398,E2 -5650.398} C_VEL
LIN {X 0,Y 502.798,Z 287.853,A -85,B 0,C 180,E1 -5652.929,E2 -5652.929} C_VEL
LIN {X 0,Y 502.832,Z 287.852,A -85,B 0,C 180,E1 -5655.427,E2 -5655.427} C_VEL
LIN {X 0,Y 502.877,Z 287.84,A -85,B 0,C 180,E1 -5658.715,E2 -5658.715} C_VEL
LIN {X 0,Y 502.851,Z 287.844,A -85,B 0,C 180,E1 -5661.964,E2 -5661.964} C_VEL
LIN {X 0,Y 502.899,Z 287.836,A -85,B 0,C 180,E1 -5664.384,E2 -5664.384} C_VEL
LIN {X 0,Y 503.012,Z 287.831,A -85,B 0,C 180,E1 -5667.595,E2 -5667.595} C_VEL
LIN {X 0,Y 503.006,Z 287.827,A -85,B 0,C 180,E1 -5669.997,E2 -5669.997} C_VEL
LIN {X 0,Y 503.012,Z 287.823,A -85,B 0,C 180,E1 -5672.4,E2 -5672.4} C_VEL
LIN {X 0,Y 502.898,Z 287.843,A -85,B 0,C 180,E1 -5675.611,E2 -5675.611} C_VEL
LIN {X 0,Y 502.871,Z 287.848,A -85,B 0,C 180,E1 -5678.031,E2 -5678.031} C_VEL
LIN {X 0,Y 502.865,Z 287.847,A -85,B 0,C 180,E1 -5681.28,E2 -5681.28} C_VEL
LIN {X 0,Y 502.884,Z 287.925,A -85,B 0,C 180,E1 -5681.907,E2 -5681.907} C_VEL
LIN {X 0,Y 503.581,Z 293.802,A -85,B 0,C 180,E1 -5683.104,E2 -5683.104} C_VEL
LIN {X 0,Y 503.287,Z 308.543,A -85,B 0,C 180,E1 -5685.99,E2 -5685.99} C_VEL
LIN {X 0,Y 503.262,Z 309.875,A -85,B 0,C 180,E1 -5686.25,E2 -5686.25} C_VEL
LIN {X 0,Y 505.448,Z 322.148,A -85,B 0,C 180,E1 -5686.509,E2 -5686.509} C_VEL
LIN {X 0,Y 504.818,Z 416.63,A -85,B 0,C 180,E1 -5687.884,E2 -5687.884} C_VEL
LIN {X 0,Y 504.693,Z 429.566,A -85,B 0,C 180,E1 -5688.229,E2 -5688.229} C_VEL
LIN {X 0,Y 504.397,Z 442.484,A -85,B 0,C 180,E1 -5688.74,E2 -5688.74} C_VEL
LIN {X 0,Y 504.049,Z 453.624,A -85,B 0,C 180,E1 -5689.334,E2 -5689.334} C_VEL
LIN {X 0,Y 503.724,Z 464.621,A -85,B 0,C 180,E1 -5690.09,E2 -5690.09} C_VEL
LIN {X 0,Y 503.364,Z 474.405,A -85,B 0,C 180,E1 -5690.923,E2 -5690.923} C_VEL
LIN {X 0,Y 503.033,Z 484.147,A -85,B 0,C 180,E1 -5691.941,E2 -5691.941} C_VEL
LIN {X 0,Y 502.776,Z 492.668,A -85,B 0,C 180,E1 -5693.037,E2 -5693.037} C_VEL
LIN {X 0,Y 502.553,Z 500.367,A -85,B 0,C 180,E1 -5694.268,E2 -5694.268} C_VEL
LIN {X 0,Y 502.339,Z 507.432,A -85,B 0,C 180,E1 -5695.698,E2 -5695.698} C_VEL
LIN {X 0,Y 502.236,Z 512.498,A -85,B 0,C 180,E1 -5697.046,E2 -5697.046} C_VEL
LIN {X 0,Y 502.088,Z 516.255,A -85,B 0,C 180,E1 -5698.414,E2 -5698.414} C_VEL
LIN {X 0,Y 502.017,Z 518.757,A -85,B 0,C 180,E1 -5699.776,E2 -5699.776} C_VEL
LIN {X 0,Y 502.001,Z 520.218,A -85,B 0,C 180,E1 -5701.35,E2 -5701.35} C_VEL
LIN {X 0,Y 502.009,Z 520.152,A -85,B 0,C 180,E1 -5702.861,E2 -5702.861} C_VEL
LIN {X 0,Y 502.037,Z 518.771,A -85,B 0,C 180,E1 -5704.316,E2 -5704.316} C_VEL
LIN {X 0,Y 502.132,Z 516.166,A -85,B 0,C 180,E1 -5705.729,E2 -5705.729} C_VEL
LIN {X 0,Y 502.205,Z 512.397,A -85,B 0,C 180,E1 -5707.091,E2 -5707.091} C_VEL
LIN {X 0,Y 502.37,Z 507.338,A -85,B 0,C 180,E1 -5708.425,E2 -5708.425} C_VEL
LIN {X 0,Y 502.535,Z 500.999,A -85,B 0,C 180,E1 -5709.719,E2 -5709.719} C_VEL
LIN {X 0,Y 502.79,Z 493.167,A -85,B 0,C 180,E1 -5710.991,E2 -5710.991} C_VEL
LIN {X 0,Y 503.058,Z 484.606,A -85,B 0,C 180,E1 -5712.105,E2 -5712.105} C_VEL
LIN {X 0,Y 503.387,Z 474.588,A -85,B 0,C 180,E1 -5713.158,E2 -5713.158} C_VEL
LIN {X 0,Y 503.758,Z 464.592,A -85,B 0,C 180,E1 -5714.009,E2 -5714.009} C_VEL
LIN {X 0,Y 504.105,Z 453.712,A -85,B 0,C 180,E1 -5714.755,E2 -5714.755} C_VEL
LIN {X 0,Y 504.431,Z 441.626,A -85,B 0,C 180,E1 -5715.393,E2 -5715.393} C_VEL
LIN {X 0,Y 504.671,Z 428.936,A -85,B 0,C 180,E1 -5715.887,E2 -5715.887} C_VEL
LIN {X 0,Y 504.882,Z 416.21,A -85,B 0,C 180,E1 -5716.215,E2 -5716.215} C_VEL
LIN {X 0,Y 505.339,Z 321.123,A -85,B 0,C 180,E1 -5717.604,E2 -5717.604} C_VEL
LIN {X 0,Y 503.235,Z 309.453,A -85,B 0,C 180,E1 -5717.862,E2 -5717.862} C_VEL
LIN {X 0,Y 503.348,Z 292.593,A -85,B 0,C 180,E1 -5720.85,E2 -5720.85} C_VEL
LIN {X 0,Y 502.828,Z 287.853,A -85,B 0,C 180,E1 -5721.744,E2 -5721.744} C_VEL
LIN {X 0,Y 502.77,Z 287.856,A -85,B 0,C 180,E1 -5725.032,E2 -5725.032} C_VEL
LIN {X 0,Y 502.746,Z 287.861,A -85,B 0,C 180,E1 -5727.913,E2 -5727.913} C_VEL
LIN {X 0,Y 502.794,Z 287.855,A -85,B 0,C 180,E1 -5730.71,E2 -5730.71} C_VEL
LIN {X 0,Y 502.835,Z 287.848,A -85,B 0,C 180,E1 -5733.432,E2 -5733.432} C_VEL
LIN {X 0,Y 502.744,Z 287.864,A -85,B 0,C 180,E1 -5736.084,E2 -5736.084} C_VEL
LIN {X 0,Y 502.732,Z 287.866,A -85,B 0,C 180,E1 -5738.686,E2 -5738.686} C_VEL
LIN {X 0,Y 502.778,Z 287.853,A -85,B 0,C 180,E1 -5741.246,E2 -5741.246} C_VEL
LIN {X 0,Y 502.769,Z 287.853,A -85,B 0,C 180,E1 -5743.765,E2 -5743.765} C_VEL
LIN {X 0,Y 502.777,Z 287.857,A -85,B 0,C 180,E1 -5746.253,E2 -5746.253} C_VEL
LIN {X 0,Y 502.828,Z 287.852,A -85,B 0,C 180,E1 -5748.716,E2 -5748.716} C_VEL
LIN {X 0,Y 502.846,Z 287.844,A -85,B 0,C 180,E1 -5751.966,E2 -5751.966} C_VEL
LIN {X 0,Y 502.889,Z 287.841,A -85,B 0,C 180,E1 -5754.386,E2 -5754.386} C_VEL
LIN {X 0,Y 502.97,Z 287.828,A -85,B 0,C 180,E1 -5757.597,E2 -5757.597} C_VEL
LIN {X 0,Y 502.966,Z 287.825,A -85,B 0,C 180,E1 -5760,E2 -5760} C_VEL
LIN {X 0,Y 502.972,Z 287.83,A -85,B 0,C 180,E1 -5762.402,E2 -5762.402} C_VEL
LIN {X 0,Y 502.907,Z 287.837,A -85,B 0,C 180,E1 -5765.614,E2 -5765.614} C_VEL
LIN {X 0,Y 502.852,Z 287.839,A -85,B 0,C 180,E1 -5768.034,E2 -5768.034} C_VEL
LIN {X 0,Y 502.849,Z 287.846,A -85,B 0,C 180,E1 -5771.284,E2 -5771.284} C_VEL
LIN {X 0,Y 502.805,Z 287.85,A -85,B 0,C 180,E1 -5774.572,E2 -5774.572} C_VEL
LIN {X 0,Y 502.812,Z 287.847,A -85,B 0,C 180,E1 -5777.909,E2 -5777.909} C_VEL
LIN {X 0,Y 502.782,Z 287.848,A -85,B 0,C 180,E1 -5780.539,E2 -5780.539} C_VEL
LIN {X 0,Y 502.776,Z 287.856,A -85,B 0,C 180,E1 -5783.041,E2 -5783.041} C_VEL
LIN {X 0,Y 502.808,Z 287.852,A -85,B 0,C 180,E1 -5785.677,E2 -5785.677} C_VEL
LIN {X 0,Y 502.799,Z 287.846,A -85,B 0,C 180,E1 -5788.375,E2 -5788.375} C_VEL
LIN {X 0,Y 502.756,Z 287.86,A -85,B 0,C 180,E1 -5791.503,E2 -5791.503} C_VEL
LIN {X 0,Y 502.768,Z 287.853,A -85,B 0,C 180,E1 -5794.448,E2 -5794.448} C_VEL
LIN {X 0,Y 502.755,Z 287.859,A -85,B 0,C 180,E1 -5797.184,E2 -5797.184} C_VEL
LIN {X 0,Y 502.812,Z 287.852,A -85,B 0,C 180,E1 -5800.013,E2 -5800.013} C_VEL
LIN {X 0,Y 502.793,Z 287.854,A -85,B 0,C 180,E1 -5802.206,E2 -5802.206} C_VEL
LIN {X 0,Y 502.77,Z 287.861,A -85,B 0,C 180,E1 -5805.472,E2 -5805.472} C_VEL
LIN {X 0,Y 502.81,Z 287.857,A -85,B 0,C 180,E1 -5807.869,E2 -5807.869} C_VEL
LIN {X 0,Y 502.797,Z 287.851,A -85,B 0,C 180,E1 -5811.03,E2 -5811.03} C_VEL
LIN {X 0,Y 502.764,Z 287.86,A -85,B 0,C 180,E1 -5814.171,E2 -5814.171} C_VEL
LIN {X 0,Y 502.813,Z 287.851,A -85,B 0,C 180,E1 -5816.997,E2 -5816.997} C_VEL
LIN {X 0,Y 502.813,Z 287.857,A -85,B 0,C 180,E1 -5820.066,E2 -5820.066} C_VEL
LIN {X 0,Y 502.821,Z 287.852,A -85,B 0,C 180,E1 -5822.538,E2 -5822.538} C_VEL
LIN {X 0,Y 502.877,Z 288.029,A -85,B 0,C 180,E1 -5825.106,E2 -5825.106} C_VEL
LIN {X 0,Y 504.413,Z 296.612,A -85,B 0,C 180,E1 -5826.571,E2 -5826.571} C_VEL
LIN {X 0,Y 504.031,Z 313.991,A -85,B 0,C 180,E1 -5829.353,E2 -5829.353} C_VEL
LIN {X 0,Y 503.478,Z 334.172,A -85,B 0,C 180,E1 -5832.539,E2 -5832.539} C_VEL
LIN {X 0,Y 503.209,Z 344.639,A -85,B 0,C 180,E1 -5834.183,E2 -5834.183} C_VEL
LIN {X 0,Y 505.379,Z 359.53,A -85,B 0,C 180,E1 -5834.477,E2 -5834.477} C_VEL
LIN {X 0,Y 504.77,Z 453.653,A -85,B 0,C 180,E1 -5835.85,E2 -5835.85} C_VEL
LIN {X 0,Y 504.442,Z 467.531,A -85,B 0,C 180,E1 -5836.226,E2 -5836.226} C_VEL
LIN {X 0,Y 504.117,Z 480.492,A -85,B 0,C 180,E1 -5836.756,E2 -5836.756} C_VEL
LIN {X 0,Y 503.864,Z 491.8,A -85,B 0,C 180,E1 -5837.384,E2 -5837.384} C_VEL
LIN {X 0,Y 503.55,Z 502.38,A -85,B 0,C 180,E1 -5838.123,E2 -5838.123} C_VEL
LIN {X 0,Y 503.181,Z 512.886,A -85,B 0,C 180,E1 -5839.033,E2 -5839.033} C_VEL
LIN {X 0,Y 502.863,Z 521.477,A -85,B 0,C 180,E1 -5839.942,E2 -5839.942} C_VEL
LIN {X 0,Y 502.624,Z 529.405,A -85,B 0,C 180,E1 -5840.953,E2 -5840.953} C_VEL
LIN {X 0,Y 502.387,Z 537.147,A -85,B 0,C 180,E1 -5842.164,E2 -5842.164} C_VEL
LIN {X 0,Y 502.224,Z 543.913,A -85,B 0,C 180,E1 -5843.494,E2 -5843.494} C_VEL
LIN {X 0,Y 502.174,Z 549.033,A -85,B 0,C 180,E1 -5844.784,E2 -5844.784} C_VEL
LIN {X 0,Y 502.138,Z 552.662,A -85,B 0,C 180,E1 -5845.99,E2 -5845.99} C_VEL
LIN {X 0,Y 502.119,Z 554.535,A -85,B 0,C 180,E1 -5846.793,E2 -5846.793} C_VEL
LIN {X 0,Y 502.091,Z 555.937,A -85,B 0,C 180,E1 -5847.596,E2 -5847.596} C_VEL
LIN {X 0,Y 501.99,Z 557.55,A -85,B 0,C 180,E1 -5849.2,E2 -5849.2} C_VEL
LIN {X 0,Y 501.983,Z 557.769,A -85,B 0,C 180,E1 -5850.003,E2 -5850.003} C_VEL
LIN {X 0,Y 502.036,Z 556.947,A -85,B 0,C 180,E1 -5851.607,E2 -5851.607} C_VEL
LIN {X 0,Y 502.092,Z 555.952,A -85,B 0,C 180,E1 -5852.409,E2 -5852.409} C_VEL
LIN {X 0,Y 502.121,Z 554.552,A -85,B 0,C 180,E1 -5853.212,E2 -5853.212} C_VEL
LIN {X 0,Y 502.102,Z 551.605,A -85,B 0,C 180,E1 -5854.418,E2 -5854.418} C_VEL
LIN {X 0,Y 502.21,Z 547.618,A -85,B 0,C 180,E1 -5855.624,E2 -5855.624} C_VEL
LIN {X 0,Y 502.332,Z 541.582,A -85,B 0,C 180,E1 -5857.014,E2 -5857.014} C_VEL
LIN {X 0,Y 502.478,Z 534.775,A -85,B 0,C 180,E1 -5858.245,E2 -5858.245} C_VEL
LIN {X 0,Y 502.715,Z 526.457,A -85,B 0,C 180,E1 -5859.457,E2 -5859.457} C_VEL
LIN {X 0,Y 502.969,Z 517.92,A -85,B 0,C 180,E1 -5860.468,E2 -5860.468} C_VEL
LIN {X 0,Y 503.413,Z 507.379,A -85,B 0,C 180,E1 -5861.477,E2 -5861.477} C_VEL
LIN {X 0,Y 503.684,Z 497.042,A -85,B 0,C 180,E1 -5862.28,E2 -5862.28} C_VEL
LIN {X 0,Y 504.042,Z 485.492,A -85,B 0,C 180,E1 -5862.995,E2 -5862.995} C_VEL
LIN {X 0,Y 504.321,Z 473.672,A -85,B 0,C 180,E1 -5863.552,E2 -5863.552} C_VEL
LIN {X 0,Y 504.678,Z 460.051,A -85,B 0,C 180,E1 -5864.004,E2 -5864.004} C_VEL
LIN {X 0,Y 504.86,Z 447.903,A -85,B 0,C 180,E1 -5864.256,E2 -5864.256} C_VEL
LIN {X 0,Y 505.315,Z 358.542,A -85,B 0,C 180,E1 -5865.542,E2 -5865.542} C_VEL
LIN {X 0,Y 503.25,Z 344.892,A -85,B 0,C 180,E1 -5865.824,E2 -5865.824} C_VEL
LIN {X 0,Y 503.802,Z 325.452,A -85,B 0,C 180,E1 -5868.927,E2 -5868.927} C_VEL
LIN {X 0,Y 504.356,Z 307.178,A -85,B 0,C 180,E1 -5871.887,E2 -5871.887} C_VEL
LIN {X 0,Y 504.603,Z 297.666,A -85,B 0,C 180,E1 -5873.449,E2 -5873.449} C_VEL
LIN {X 0,Y 502.866,Z 287.848,A -85,B 0,C 180,E1 -5875.201,E2 -5875.201} C_VEL
LIN {X 0,Y 502.845,Z 287.851,A -85,B 0,C 180,E1 -5878.295,E2 -5878.295} C_VEL
LIN {X 0,Y 502.797,Z 287.852,A -85,B 0,C 180,E1 -5881.499,E2 -5881.499} C_VEL
LIN {X 0,Y 502.807,Z 287.854,A -85,B 0,C 180,E1 -5883.994,E2 -5883.994} C_VEL
LIN {X 0,Y 502.779,Z 287.851,A -85,B 0,C 180,E1 -5887.178,E2 -5887.178} C_VEL
LIN {X 0,Y 502.789,Z 287.855,A -85,B 0,C 180,E1 -5890.015,E2 -5890.015} C_VEL
LIN {X 0,Y 502.804,Z 287.855,A -85,B 0,C 180,E1 -5892.199,E2 -5892.199} C_VEL
LIN {X 0,Y 502.785,Z 287.85,A -85,B 0,C 180,E1 -5895.47,E2 -5895.47} C_VEL
LIN {X 0,Y 502.819,Z 287.849,A -85,B 0,C 180,E1 -5898.934,E2 -5898.934} C_VEL
LIN {X 0,Y 502.79,Z 287.852,A -85,B 0,C 180,E1 -5902.046,E2 -5902.046} C_VEL
LIN {X 0,Y 502.803,Z 287.852,A -85,B 0,C 180,E1 -5905.034,E2 -5905.034} C_VEL
LIN {X 0,Y 502.783,Z 287.851,A -85,B 0,C 180,E1 -5907.915,E2 -5907.915} C_VEL
LIN {X 0,Y 502.821,Z 287.854,A -85,B 0,C 180,E1 -5910.712,E2 -5910.712} C_VEL
LIN {X 0,Y 502.857,Z 287.843,A -85,B 0,C 180,E1 -5913.439,E2 -5913.439} C_VEL
LIN {X 0,Y 502.783,Z 287.851,A -85,B 0,C 180,E1 -5916.086,E2 -5916.086} C_VEL
LIN {X 0,Y 502.774,Z 287.856,A -85,B 0,C 180,E1 -5918.688,E2 -5918.688} C_VEL
LIN {X 0,Y 502.82,Z 287.852,A -85,B 0,C 180,E1 -5921.248,E2 -5921.248} C_VEL
LIN {X 0,Y 502.81,Z 287.848,A -85,B 0,C 180,E1 -5923.767,E2 -5923.767} C_VEL
LIN {X 0,Y 502.819,Z 287.846,A -85,B 0,C 180,E1 -5926.254,E2 -5926.254} C_VEL
LIN {X 0,Y 502.867,Z 287.842,A -85,B 0,C 180,E1 -5928.717,E2 -5928.717} C_VEL
LIN {X 0,Y 502.89,Z 287.838,A -85,B 0,C 180,E1 -5931.966,E2 -5931.966} C_VEL
LIN {X 0,Y 502.921,Z 287.833,A -85,B 0,C 180,E1 -5934.386,E2 -5934.386} C_VEL
LIN {X 0,Y 503.01,Z 287.829,A -85,B 0,C 180,E1 -5937.598,E2 -5937.598} C_VEL
LIN {X 0,Y 503.009,Z 287.825,A -85,B 0,C 180,E1 -5940,E2 -5940} C_VEL
LIN {X 0,Y 503.008,Z 287.823,A -85,B 0,C 180,E1 -5942.402,E2 -5942.402} C_VEL
LIN {X 0,Y 502.912,Z 287.844,A -85,B 0,C 180,E1 -5945.614,E2 -5945.614} C_VEL
LIN {X 0,Y 502.854,Z 287.842,A -85,B 0,C 180,E1 -5948.844,E2 -5948.844} C_VEL
LIN {X 0,Y 502.834,Z 287.848,A -85,B 0,C 180,E1 -5952.102,E2 -5952.102} C_VEL
LIN {X 0,Y 502.839,Z 287.846,A -85,B 0,C 180,E1 -5955.4,E2 -5955.4} C_VEL
LIN {X 0,Y 502.811,Z 287.847,A -85,B 0,C 180,E1 -5958.753,E2 -5958.753} C_VEL
LIN {X 0,Y 502.769,Z 287.853,A -85,B 0,C 180,E1 -5961.312,E2 -5961.312} C_VEL
LIN {X 0,Y 502.758,Z 287.861,A -85,B 0,C 180,E1 -5963.916,E2 -5963.916} C_VEL
LIN {X 0,Y 502.775,Z 287.854,A -85,B 0,C 180,E1 -5966.571,E2 -5966.571} C_VEL
LIN {X 0,Y 502.803,Z 287.853,A -85,B 0,C 180,E1 -5969.934,E2 -5969.934} C_VEL
LIN {X 0,Y 502.797,Z 287.849,A -85,B 0,C 180,E1 -5973.034,E2 -5973.034} C_VEL
LIN {X 0,Y 502.739,Z 287.86,A -85,B 0,C 180,E1 -5975.954,E2 -5975.954} C_VEL
LIN {X 0,Y 502.766,Z 287.854,A -85,B 0,C 180,E1 -5978.98,E2 -5978.98} C_VEL
LIN {X 0,Y 502.743,Z 287.86,A -85,B 0,C 180,E1 -5982.192,E2 -5982.192} C_VEL
LIN {X 0,Y 502.776,Z 287.851,A -85,B 0,C 180,E1 -5985.471,E2 -5985.471} C_VEL
LIN {X 0,Y 502.749,Z 287.86,A -85,B 0,C 180,E1 -5988.927,E2 -5988.927} C_VEL
LIN {X 0,Y 502.742,Z 287.857,A -85,B 0,C 180,E1 -5992.041,E2 -5992.041} C_VEL
LIN {X 0,Y 502.705,Z 287.866,A -85,B 0,C 180,E1 -5995.026,E2 -5995.026} C_VEL
LIN {X 0,Y 502.749,Z 287.859,A -85,B 0,C 180,E1 -5997.202,E2 -5997.202} C_VEL
LIN {X 0,Y 502.066,Z 287.942,A -85,B 0,C 180,E1 -5997.871,E2 -5997.871} C_VEL
LIN {X 0,Y 499.199,Z 288.306,A -85,B 0,C 180,E1 -5998.957,E2 -5998.957} C_VEL
LIN {X 0,Y 496.788,Z 288.601,A -85,B 0,C 180,E1 -5999.832,E2 -5999.832} C_VEL
LIN {X 0,Y 495.761,Z 288.728,A -85,B 0,C 180,E1 -6000.508,E2 -6000.508} C_VEL
LIN {X 0,Y 495.681,Z 288.737,A -85,B 0,C 180,E1 -6000.737,E2 -6000.737} C_VEL
LIN {X 0,Y 495.724,Z 288.735,A -85,B 0,C 180,E1 -6003.274,E2 -6003.274} C_VEL
LIN {X 0,Y 495.706,Z 288.733,A -85,B 0,C 180,E1 -6005.721,E2 -6005.721} C_VEL
LIN {X 0,Y 495.745,Z 288.728,A -85,B 0,C 180,E1 -6008.37,E2 -6008.37} C_VEL
LIN {X 0,Y 495.769,Z 288.73,A -85,B 0,C 180,E1 -6010.97,E2 -6010.97} C_VEL
LIN {X 0,Y 495.828,Z 288.718,A -85,B 0,C 180,E1 -6014.548,E2 -6014.548} C_VEL
LIN {X 0,Y 495.834,Z 288.717,A -85,B 0,C 180,E1 -6017.964,E2 -6017.964} C_VEL
LIN {X 0,Y 495.799,Z 288.724,A -85,B 0,C 180,E1 -6021.027,E2 -6021.027} C_VEL
LIN {X 0,Y 495.824,Z 288.727,A -85,B 0,C 180,E1 -6023.487,E2 -6023.487} C_VEL
LIN {X 0,Y 495.706,Z 288.736,A -85,B 0,C 180,E1 -6025.933,E2 -6025.933} C_VEL
LIN {X 0,Y 495.979,Z 288.708,A -85,B 0,C 180,E1 -6027.561,E2 -6027.561} C_VEL
LIN {X 0,Y 495.975,Z 288.702,A -85,B 0,C 180,E1 -6029.997,E2 -6029.997} C_VEL
LIN {X 0,Y 495.979,Z 288.699,A -85,B 0,C 180,E1 -6032.434,E2 -6032.434} C_VEL
LIN {X 0,Y 495.856,Z 288.722,A -85,B 0,C 180,E1 -6035.691,E2 -6035.691} C_VEL
LIN {X 0,Y 495.829,Z 288.724,A -85,B 0,C 180,E1 -6038.145,E2 -6038.145} C_VEL
LIN {X 0,Y 495.841,Z 288.834,A -85,B 0,C 180,E1 -6041.769,E2 -6041.769} C_VEL
LIN {X 0,Y 496.612,Z 295.222,A -85,B 0,C 180,E1 -6043.083,E2 -6043.083} C_VEL
LIN {X 0,Y 496.291,Z 310.09,A -85,B 0,C 180,E1 -6046.026,E2 -6046.026} C_VEL
LIN {X 0,Y 498.631,Z 322.283,A -85,B 0,C 180,E1 -6046.29,E2 -6046.29} C_VEL
LIN {X 0,Y 497.947,Z 416.875,A -85,B 0,C 180,E1 -6047.687,E2 -6047.687} C_VEL
LIN {X 0,Y 497.798,Z 429.84,A -85,B 0,C 180,E1 -6048.038,E2 -6048.038} C_VEL
LIN {X 0,Y 497.505,Z 442.513,A -85,B 0,C 180,E1 -6048.545,E2 -6048.545} C_VEL
LIN {X 0,Y 497.111,Z 454.324,A -85,B 0,C 180,E1 -6049.186,E2 -6049.186} C_VEL
LIN {X 0,Y 496.769,Z 465.233,A -85,B 0,C 180,E1 -6049.952,E2 -6049.952} C_VEL
LIN {X 0,Y 496.355,Z 476.56,A -85,B 0,C 180,E1 -6050.951,E2 -6050.951} C_VEL
LIN {X 0,Y 495.967,Z 486.484,A -85,B 0,C 180,E1 -6052.052,E2 -6052.052} C_VEL
LIN {X 0,Y 495.719,Z 494.1,A -85,B 0,C 180,E1 -6053.088,E2 -6053.088} C_VEL
LIN {X 0,Y 495.501,Z 501.301,A -85,B 0,C 180,E1 -6054.283,E2 -6054.283} C_VEL
LIN {X 0,Y 495.286,Z 507.826,A -85,B 0,C 180,E1 -6055.64,E2 -6055.64} C_VEL
LIN {X 0,Y 495.168,Z 512.852,A -85,B 0,C 180,E1 -6057.007,E2 -6057.007} C_VEL
LIN {X 0,Y 495.011,Z 516.437,A -85,B 0,C 180,E1 -6058.326,E2 -6058.326} C_VEL
LIN {X 0,Y 494.941,Z 519.347,A -85,B 0,C 180,E1 -6059.982,E2 -6059.982} C_VEL
LIN {X 0,Y 494.922,Z 520.121,A -85,B 0,C 180,E1 -6060.739,E2 -6060.739} C_VEL
LIN {X 0,Y 494.903,Z 520.571,A -85,B 0,C 180,E1 -6061.692,E2 -6061.692} C_VEL
LIN {X 0,Y 494.913,Z 520.292,A -85,B 0,C 180,E1 -6063.088,E2 -6063.088} C_VEL
LIN {X 0,Y 494.947,Z 518.688,A -85,B 0,C 180,E1 -6064.604,E2 -6064.604} C_VEL
LIN {X 0,Y 495.083,Z 515.963,A -85,B 0,C 180,E1 -6065.987,E2 -6065.987} C_VEL
LIN {X 0,Y 495.15,Z 511.996,A -85,B 0,C 180,E1 -6067.359,E2 -6067.359} C_VEL
LIN {X 0,Y 495.294,Z 506.792,A -85,B 0,C 180,E1 -6068.7,E2 -6068.7} C_VEL
LIN {X 0,Y 495.511,Z 500.264,A -85,B 0,C 180,E1 -6070.013,E2 -6070.013} C_VEL
LIN {X 0,Y 495.745,Z 493.235,A -85,B 0,C 180,E1 -6071.148,E2 -6071.148} C_VEL
LIN {X 0,Y 496.093,Z 484.535,A -85,B 0,C 180,E1 -6072.285,E2 -6072.285} C_VEL
LIN {X 0,Y 496.449,Z 474.45,A -85,B 0,C 180,E1 -6073.354,E2 -6073.354} C_VEL
LIN {X 0,Y 496.855,Z 463.391,A -85,B 0,C 180,E1 -6074.292,E2 -6074.292} C_VEL
LIN {X 0,Y 497.279,Z 451.628,A -85,B 0,C 180,E1 -6075.071,E2 -6075.071} C_VEL
LIN {X 0,Y 497.595,Z 439.85,A -85,B 0,C 180,E1 -6075.674,E2 -6075.674} C_VEL
LIN {X 0,Y 497.869,Z 426.948,A -85,B 0,C 180,E1 -6076.152,E2 -6076.152} C_VEL
LIN {X 0,Y 498.013,Z 413.581,A -85,B 0,C 180,E1 -6076.465,E2 -6076.465} C_VEL
LIN {X 0,Y 498.631,Z 322.587,A -85,B 0,C 180,E1 -6077.802,E2 -6077.802} C_VEL
LIN {X 0,Y 496.248,Z 309.742,A -85,B 0,C 180,E1 -6078.082,E2 -6078.082} C_VEL
LIN {X 0,Y 496.372,Z 294.299,A -85,B 0,C 180,E1 -6080.835,E2 -6080.835} C_VEL
LIN {X 0,Y 495.821,Z 288.971,A -85,B 0,C 180,E1 -6081.803,E2 -6081.803} C_VEL
LIN {X 0,Y 495.772,Z 288.733,A -85,B 0,C 180,E1 -6081.928,E2 -6081.928} C_VEL
LIN {X 0,Y 495.745,Z 288.731,A -85,B 0,C 180,E1 -6085.454,E2 -6085.454} C_VEL
LIN {X 0,Y 495.717,Z 288.739,A -85,B 0,C 180,E1 -6088.361,E2 -6088.361} C_VEL
LIN {X 0,Y 495.745,Z 288.73,A -85,B 0,C 180,E1 -6091.503,E2 -6091.503} C_VEL
LIN {X 0,Y 495.754,Z 288.733,A -85,B 0,C 180,E1 -6093.93,E2 -6093.93} C_VEL
LIN {X 0,Y 495.712,Z 288.736,A -85,B 0,C 180,E1 -6097.136,E2 -6097.136} C_VEL
LIN {X 0,Y 495.72,Z 288.737,A -85,B 0,C 180,E1 -6100.107,E2 -6100.107} C_VEL
LIN {X 0,Y 495.734,Z 288.737,A -85,B 0,C 180,E1 -6102.679,E2 -6102.679} C_VEL
LIN {X 0,Y 495.736,Z 288.731,A -85,B 0,C 180,E1 -6105.215,E2 -6105.215} C_VEL
LIN {X 0,Y 495.801,Z 288.729,A -85,B 0,C 180,E1 -6108.554,E2 -6108.554} C_VEL
LIN {X 0,Y 495.818,Z 288.719,A -85,B 0,C 180,E1 -6111.851,E2 -6111.851} C_VEL
LIN {X 0,Y 495.843,Z 288.718,A -85,B 0,C 180,E1 -6114.306,E2 -6114.306} C_VEL
LIN {X 0,Y 495.94,Z 288.704,A -85,B 0,C 180,E1 -6117.563,E2 -6117.563} C_VEL
LIN {X 0,Y 495.938,Z 288.7,A -85,B 0,C 180,E1 -6120,E2 -6120} C_VEL
LIN {X 0,Y 495.942,Z 288.706,A -85,B 0,C 180,E1 -6122.437,E2 -6122.437} C_VEL
LIN {X 0,Y 495.861,Z 288.714,A -85,B 0,C 180,E1 -6125.694,E2 -6125.694} C_VEL
LIN {X 0,Y 495.825,Z 288.715,A -85,B 0,C 180,E1 -6128.149,E2 -6128.149} C_VEL
LIN {X 0,Y 495.822,Z 288.719,A -85,B 0,C 180,E1 -6131.446,E2 -6131.446} C_VEL
LIN {X 0,Y 495.748,Z 288.731,A -85,B 0,C 180,E1 -6134.784,E2 -6134.784} C_VEL
LIN {X 0,Y 495.741,Z 288.735,A -85,B 0,C 180,E1 -6137.32,E2 -6137.32} C_VEL
LIN {X 0,Y 495.73,Z 288.727,A -85,B 0,C 180,E1 -6139.892,E2 -6139.892} C_VEL
LIN {X 0,Y 495.743,Z 288.73,A -85,B 0,C 180,E1 -6142.872,E2 -6142.872} C_VEL
LIN {X 0,Y 495.76,Z 288.726,A -85,B 0,C 180,E1 -6146.07,E2 -6146.07} C_VEL
LIN {X 0,Y 495.737,Z 288.727,A -85,B 0,C 180,E1 -6148.817,E2 -6148.817} C_VEL
LIN {X 0,Y 495.719,Z 288.735,A -85,B 0,C 180,E1 -6151.73,E2 -6151.73} C_VEL
LIN {X 0,Y 495.739,Z 288.728,A -85,B 0,C 180,E1 -6154.699,E2 -6154.699} C_VEL
LIN {X 0,Y 495.706,Z 288.74,A -85,B 0,C 180,E1 -6157.564,E2 -6157.564} C_VEL
LIN {X 0,Y 495.777,Z 288.728,A -85,B 0,C 180,E1 -6160.058,E2 -6160.058} C_VEL
LIN {X 0,Y 495.731,Z 288.732,A -85,B 0,C 180,E1 -6162.883,E2 -6162.883} C_VEL
LIN {X 0,Y 495.706,Z 288.74,A -85,B 0,C 180,E1 -6166.003,E2 -6166.003} C_VEL
LIN {X 0,Y 495.746,Z 288.73,A -85,B 0,C 180,E1 -6168.709,E2 -6168.709} C_VEL
LIN {X 0,Y 495.74,Z 288.733,A -85,B 0,C 180,E1 -6171.414,E2 -6171.414} C_VEL
LIN {X 0,Y 495.737,Z 288.733,A -85,B 0,C 180,E1 -6174.467,E2 -6174.467} C_VEL
LIN {X 0,Y 495.75,Z 288.733,A -85,B 0,C 180,E1 -6177.41,E2 -6177.41} C_VEL
LIN {X 0,Y 495.765,Z 288.734,A -85,B 0,C 180,E1 -6180.259,E2 -6180.259} C_VEL
LIN {X 0,Y 495.82,Z 288.723,A -85,B 0,C 180,E1 -6183.252,E2 -6183.252} C_VEL
LIN {X 0,Y 495.831,Z 288.904,A -85,B 0,C 180,E1 -6184.928,E2 -6184.928} C_VEL
LIN {X 0,Y 497.468,Z 297.986,A -85,B 0,C 180,E1 -6186.505,E2 -6186.505} C_VEL
LIN {X 0,Y 497.037,Z 315.234,A -85,B 0,C 180,E1 -6189.303,E2 -6189.303} C_VEL
LIN {X 0,Y 496.472,Z 335.193,A -85,B 0,C 180,E1 -6192.498,E2 -6192.498} C_VEL
LIN {X 0,Y 496.229,Z 344.38,A -85,B 0,C 180,E1 -6193.958,E2 -6193.958} C_VEL
LIN {X 0,Y 498.509,Z 360.001,A -85,B 0,C 180,E1 -6194.268,E2 -6194.268} C_VEL
LIN {X 0,Y 497.896,Z 453.302,A -85,B 0,C 180,E1 -6195.65,E2 -6195.65} C_VEL
LIN {X 0,Y 497.56,Z 467.197,A -85,B 0,C 180,E1 -6196.032,E2 -6196.032} C_VEL
LIN {X 0,Y 497.215,Z 480.173,A -85,B 0,C 180,E1 -6196.569,E2 -6196.569} C_VEL
LIN {X 0,Y 496.91,Z 491.944,A -85,B 0,C 180,E1 -6197.234,E2 -6197.234} C_VEL
LIN {X 0,Y 496.539,Z 503.37,A -85,B 0,C 180,E1 -6198.057,E2 -6198.057} C_VEL
LIN {X 0,Y 496.142,Z 513.641,A -85,B 0,C 180,E1 -6198.979,E2 -6198.979} C_VEL
LIN {X 0,Y 495.795,Z 522.876,A -85,B 0,C 180,E1 -6200.003,E2 -6200.003} C_VEL
LIN {X 0,Y 495.491,Z 531.872,A -85,B 0,C 180,E1 -6201.233,E2 -6201.233} C_VEL
LIN {X 0,Y 495.274,Z 539.115,A -85,B 0,C 180,E1 -6202.461,E2 -6202.461} C_VEL
LIN {X 0,Y 495.122,Z 545.191,A -85,B 0,C 180,E1 -6203.761,E2 -6203.761} C_VEL
LIN {X 0,Y 495.035,Z 550.078,A -85,B 0,C 180,E1 -6205.117,E2 -6205.117} C_VEL
LIN {X 0,Y 495.032,Z 552.39,A -85,B 0,C 180,E1 -6205.932,E2 -6205.932} C_VEL
LIN {X 0,Y 495.041,Z 554.266,A -85,B 0,C 180,E1 -6206.747,E2 -6206.747} C_VEL
LIN {X 0,Y 494.997,Z 555.67,A -85,B 0,C 180,E1 -6207.562,E2 -6207.562} C_VEL
LIN {X 0,Y 494.962,Z 556.673,A -85,B 0,C 180,E1 -6208.375,E2 -6208.375} C_VEL
LIN {X 0,Y 494.901,Z 557.506,A -85,B 0,C 180,E1 -6210.003,E2 -6210.003} C_VEL
LIN {X 0,Y 494.962,Z 556.685,A -85,B 0,C 180,E1 -6211.63,E2 -6211.63} C_VEL
LIN {X 0,Y 494.998,Z 555.689,A -85,B 0,C 180,E1 -6212.444,E2 -6212.444} C_VEL
LIN {X 0,Y 495.042,Z 554.288,A -85,B 0,C 180,E1 -6213.258,E2 -6213.258} C_VEL
LIN {X 0,Y 495.008,Z 551.34,A -85,B 0,C 180,E1 -6214.481,E2 -6214.481} C_VEL
LIN {X 0,Y 495.127,Z 547.352,A -85,B 0,C 180,E1 -6215.705,E2 -6215.705} C_VEL
LIN {X 0,Y 495.258,Z 541.21,A -85,B 0,C 180,E1 -6217.135,E2 -6217.135} C_VEL
LIN {X 0,Y 495.424,Z 534.502,A -85,B 0,C 180,E1 -6218.363,E2 -6218.363} C_VEL
LIN {X 0,Y 495.679,Z 526.18,A -85,B 0,C 180,E1 -6219.592,E2 -6219.592} C_VEL
LIN {X 0,Y 495.968,Z 517.638,A -85,B 0,C 180,E1 -6220.617,E2 -6220.617} C_VEL
LIN {X 0,Y 496.432,Z 507.092,A -85,B 0,C 180,E1 -6221.64,E2 -6221.64} C_VEL
LIN {X 0,Y 496.755,Z 495.777,A -85,B 0,C 180,E1 -6222.525,E2 -6222.525} C_VEL
LIN {X 0,Y 497.095,Z 485.188,A -85,B 0,C 180,E1 -6223.18,E2 -6223.18} C_VEL
LIN {X 0,Y 497.413,Z 473.349,A -85,B 0,C 180,E1 -6223.743,E2 -6223.743} C_VEL
LIN {X 0,Y 497.779,Z 459.699,A -85,B 0,C 180,E1 -6224.202,E2 -6224.202} C_VEL
LIN {X 0,Y 497.992,Z 445.77,A -85,B 0,C 180,E1 -6224.483,E2 -6224.483} C_VEL
LIN {X 0,Y 498.434,Z 358.998,A -85,B 0,C 180,E1 -6225.751,E2 -6225.751} C_VEL
LIN {X 0,Y 496.259,Z 344.731,A -85,B 0,C 180,E1 -6226.037,E2 -6226.037} C_VEL
LIN {X 0,Y 496.857,Z 325.21,A -85,B 0,C 180,E1 -6229.202,E2 -6229.202} C_VEL
LIN {X 0,Y 497.4,Z 308.243,A -85,B 0,C 180,E1 -6231.99,E2 -6231.99} C_VEL
LIN {X 0,Y 497.681,Z 299.227,A -85,B 0,C 180,E1 -6233.49,E2 -6233.49} C_VEL
LIN {X 0,Y 495.827,Z 288.725,A -85,B 0,C 180,E1 -6235.391,E2 -6235.391} C_VEL
LIN {X 0,Y 495.79,Z 288.728,A -85,B 0,C 180,E1 -6238.493,E2 -6238.493} C_VEL
LIN {X 0,Y 495.759,Z 288.731,A -85,B 0,C 180,E1 -6241.725,E2 -6241.725} C_VEL
LIN {X 0,Y 495.771,Z 288.726,A -85,B 0,C 180,E1 -6244.694,E2 -6244.694} C_VEL
LIN {X 0,Y 495.731,Z 288.73,A -85,B 0,C 180,E1 -6247.562,E2 -6247.562} C_VEL
LIN {X 0,Y 495.768,Z 288.728,A -85,B 0,C 180,E1 -6250.7,E2 -6250.7} C_VEL
LIN {X 0,Y 495.728,Z 288.733,A -85,B 0,C 180,E1 -6254.001,E2 -6254.001} C_VEL
LIN {X 0,Y 495.725,Z 288.731,A -85,B 0,C 180,E1 -6257.117,E2 -6257.117} C_VEL
LIN {X 0,Y 495.757,Z 288.727,A -85,B 0,C 180,E1 -6259.953,E2 -6259.953} C_VEL
LIN {X 0,Y 495.727,Z 288.738,A -85,B 0,C 180,E1 -6262.553,E2 -6262.553} C_VEL
LIN {X 0,Y 495.778,Z 288.723,A -85,B 0,C 180,E1 -6265.457,E2 -6265.457} C_VEL
LIN {X 0,Y 495.754,Z 288.73,A -85,B 0,C 180,E1 -6268.364,E2 -6268.364} C_VEL
LIN {X 0,Y 495.783,Z 288.723,A -85,B 0,C 180,E1 -6271.506,E2 -6271.506} C_VEL
LIN {X 0,Y 495.785,Z 288.722,A -85,B 0,C 180,E1 -6273.932,E2 -6273.932} C_VEL
LIN {X 0,Y 495.753,Z 288.732,A -85,B 0,C 180,E1 -6277.139,E2 -6277.139} C_VEL
LIN {X 0,Y 495.762,Z 288.725,A -85,B 0,C 180,E1 -6280.109,E2 -6280.109} C_VEL
LIN {X 0,Y 495.771,Z 288.727,A -85,B 0,C 180,E1 -6282.681,E2 -6282.681} C_VEL
LIN {X 0,Y 495.779,Z 288.731,A -85,B 0,C 180,E1 -6285.217,E2 -6285.217} C_VEL
LIN {X 0,Y 495.841,Z 288.716,A -85,B 0,C 180,E1 -6288.555,E2 -6288.555} C_VEL
LIN {X 0,Y 495.862,Z 288.714,A -85,B 0,C 180,E1 -6291.852,E2 -6291.852} C_VEL
LIN {X 0,Y 495.877,Z 288.711,A -85,B 0,C 180,E1 -6294.306,E2 -6294.306} C_VEL
LIN {X 0,Y 495.979,Z 288.705,A -85,B 0,C 180,E1 -6297.564,E2 -6297.564} C_VEL
LIN {X 0,Y 495.981,Z 288.7,A -85,B 0,C 180,E1 -6300,E2 -6300} C_VEL
LIN {X 0,Y 495.977,Z 288.698,A -85,B 0,C 180,E1 -6302.436,E2 -6302.436} C_VEL
LIN {X 0,Y 495.868,Z 288.72,A -85,B 0,C 180,E1 -6305.694,E2 -6305.694} C_VEL
LIN {X 0,Y 495.825,Z 288.718,A -85,B 0,C 180,E1 -6308.97,E2 -6308.97} C_VEL
LIN {X 0,Y 495.818,Z 288.723,A -85,B 0,C 180,E1 -6312.035,E2 -6312.035} C_VEL
LIN {X 0,Y 495.814,Z 288.722,A -85,B 0,C 180,E1 -6315.451,E2 -6315.451} C_VEL
LIN {X 0,Y 495.766,Z 288.725,A -85,B 0,C 180,E1 -6319.029,E2 -6319.029} C_VEL
LIN {X 0,Y 495.73,Z 288.733,A -85,B 0,C 180,E1 -6321.63,E2 -6321.63} C_VEL
LIN {X 0,Y 495.704,Z 288.738,A -85,B 0,C 180,E1 -6324.278,E2 -6324.278} C_VEL
LIN {X 0,Y 495.721,Z 288.73,A -85,B 0,C 180,E1 -6326.98,E2 -6326.98} C_VEL
LIN {X 0,Y 495.752,Z 288.735,A -85,B 0,C 180,E1 -6330.146,E2 -6330.146} C_VEL
LIN {X 0,Y 495.746,Z 288.727,A -85,B 0,C 180,E1 -6333.237,E2 -6333.237} C_VEL
LIN {X 0,Y 495.681,Z 288.74,A -85,B 0,C 180,E1 -6336.083,E2 -6336.083} C_VEL
LIN {X 0,Y 495.726,Z 288.734,A -85,B 0,C 180,E1 -6338.764,E2 -6338.764} C_VEL
LIN {X 0,Y 495.699,Z 288.734,A -85,B 0,C 180,E1 -6341.787,E2 -6341.787} C_VEL
LIN {X 0,Y 495.729,Z 288.731,A -85,B 0,C 180,E1 -6345.142,E2 -6345.142} C_VEL
LIN {X 0,Y 495.698,Z 288.736,A -85,B 0,C 180,E1 -6348.213,E2 -6348.213} C_VEL
LIN {X 0,Y 495.705,Z 288.733,A -85,B 0,C 180,E1 -6351.404,E2 -6351.404} C_VEL
LIN {X 0,Y 495.655,Z 288.743,A -85,B 0,C 180,E1 -6354.454,E2 -6354.454} C_VEL
LIN {X 0,Y 495.72,Z 288.732,A -85,B 0,C 180,E1 -6357.402,E2 -6357.402} C_VEL
LIN {X 0,Y 495.697,Z 288.734,A -85,B 0,C 180,E1 -6360.248,E2 -6360.248} C_VEL
LIN {X 0,Y 495.681,Z 288.737,A -85,B 0,C 180,E1 -6360.737,E2 -6360.737} C_VEL
LIN {X 0,Y 495.02,Z 288.822,A -85,B 0,C 180,E1 -6361.416,E2 -6361.416} C_VEL
LIN {X 0,Y 492.158,Z 289.177,A -85,B 0,C 180,E1 -6362.518,E2 -6362.518} C_VEL
LIN {X 0,Y 489.744,Z 289.478,A -85,B 0,C 180,E1 -6363.407,E2 -6363.407} C_VEL
LIN {X 0,Y 488.723,Z 289.602,A -85,B 0,C 180,E1 -6364.093,E2 -6364.093} C_VEL
LIN {X 0,Y 488.648,Z 289.612,A -85,B 0,C 180,E1 -6364.325,E2 -6364.325} C_VEL
LIN {X 0,Y 488.725,Z 289.61,A -85,B 0,C 180,E1 -6367.152,E2 -6367.152} C_VEL
LIN {X 0,Y 488.723,Z 289.603,A -85,B 0,C 180,E1 -6369.809,E2 -6369.809} C_VEL
LIN {X 0,Y 488.695,Z 289.606,A -85,B 0,C 180,E1 -6372.42,E2 -6372.42} C_VEL
LIN {X 0,Y 488.759,Z 289.603,A -85,B 0,C 180,E1 -6374.998,E2 -6374.998} C_VEL
LIN {X 0,Y 488.809,Z 289.591,A -85,B 0,C 180,E1 -6378.386,E2 -6378.386} C_VEL
LIN {X 0,Y 488.762,Z 289.602,A -85,B 0,C 180,E1 -6381.731,E2 -6381.731} C_VEL
LIN {X 0,Y 488.817,Z 289.591,A -85,B 0,C 180,E1 -6384.222,E2 -6384.222} C_VEL
LIN {X 0,Y 488.945,Z 289.583,A -85,B 0,C 180,E1 -6387.526,E2 -6387.526} C_VEL
LIN {X 0,Y 488.944,Z 289.578,A -85,B 0,C 180,E1 -6389.997,E2 -6389.997} C_VEL
LIN {X 0,Y 488.945,Z 289.575,A -85,B 0,C 180,E1 -6392.469,E2 -6392.469} C_VEL
LIN {X 0,Y 488.816,Z 289.6,A -85,B 0,C 180,E1 -6395.773,E2 -6395.773} C_VEL
LIN {X 0,Y 488.778,Z 289.601,A -85,B 0,C 180,E1 -6398.264,E2 -6398.264} C_VEL
LIN {X 0,Y 488.82,Z 289.648,A -85,B 0,C 180,E1 -6401.609,E2 -6401.609} C_VEL
LIN {X 0,Y 489.636,Z 296.643,A -85,B 0,C 180,E1 -6403.062,E2 -6403.062} C_VEL
LIN {X 0,Y 489.324,Z 310.281,A -85,B 0,C 180,E1 -6405.782,E2 -6405.782} C_VEL
LIN {X 0,Y 491.743,Z 322.883,A -85,B 0,C 180,E1 -6406.072,E2 -6406.072} C_VEL
LIN {X 0,Y 491.083,Z 417.075,A -85,B 0,C 180,E1 -6407.486,E2 -6407.486} C_VEL
LIN {X 0,Y 490.917,Z 430.068,A -85,B 0,C 180,E1 -6407.842,E2 -6407.842} C_VEL
LIN {X 0,Y 490.619,Z 441.794,A -85,B 0,C 180,E1 -6408.311,E2 -6408.311} C_VEL
LIN {X 0,Y 490.234,Z 453.839,A -85,B 0,C 180,E1 -6408.96,E2 -6408.96} C_VEL
LIN {X 0,Y 489.849,Z 464.463,A -85,B 0,C 180,E1 -6409.7,E2 -6409.7} C_VEL
LIN {X 0,Y 489.452,Z 474.74,A -85,B 0,C 180,E1 -6410.593,E2 -6410.593} C_VEL
LIN {X 0,Y 489.126,Z 483.226,A -85,B 0,C 180,E1 -6411.489,E2 -6411.489} C_VEL
LIN {X 0,Y 488.849,Z 491.973,A -85,B 0,C 180,E1 -6412.613,E2 -6412.613} C_VEL
LIN {X 0,Y 488.52,Z 499.226,A -85,B 0,C 180,E1 -6413.75,E2 -6413.75} C_VEL
LIN {X 0,Y 488.3,Z 505.403,A -85,B 0,C 180,E1 -6414.94,E2 -6414.94} C_VEL
LIN {X 0,Y 488.183,Z 510.014,A -85,B 0,C 180,E1 -6416.041,E2 -6416.041} C_VEL
LIN {X 0,Y 488.023,Z 514.606,A -85,B 0,C 180,E1 -6417.436,E2 -6417.436} C_VEL
LIN {X 0,Y 487.92,Z 517.23,A -85,B 0,C 180,E1 -6418.52,E2 -6418.52} C_VEL
LIN {X 0,Y 487.86,Z 518.725,A -85,B 0,C 180,E1 -6419.322,E2 -6419.322} C_VEL
LIN {X 0,Y 487.848,Z 519.959,A -85,B 0,C 180,E1 -6420.274,E2 -6420.274} C_VEL
LIN {X 0,Y 487.805,Z 520.855,A -85,B 0,C 180,E1 -6421.784,E2 -6421.784} C_VEL
LIN {X 0,Y 487.824,Z 520.432,A -85,B 0,C 180,E1 -6423.322,E2 -6423.322} C_VEL
LIN {X 0,Y 487.862,Z 518.695,A -85,B 0,C 180,E1 -6424.802,E2 -6424.802} C_VEL
LIN {X 0,Y 488.002,Z 515.716,A -85,B 0,C 180,E1 -6426.245,E2 -6426.245} C_VEL
LIN {X 0,Y 488.107,Z 511.584,A -85,B 0,C 180,E1 -6427.635,E2 -6427.635} C_VEL
LIN {X 0,Y 488.284,Z 506.213,A -85,B 0,C 180,E1 -6428.992,E2 -6428.992} C_VEL
LIN {X 0,Y 488.522,Z 499.349,A -85,B 0,C 180,E1 -6430.338,E2 -6430.338} C_VEL
LIN {X 0,Y 488.825,Z 491.133,A -85,B 0,C 180,E1 -6431.615,E2 -6431.615} C_VEL
LIN {X 0,Y 489.184,Z 482.652,A -85,B 0,C 180,E1 -6432.685,E2 -6432.685} C_VEL
LIN {X 0,Y 489.599,Z 472.74,A -85,B 0,C 180,E1 -6433.703,E2 -6433.703} C_VEL
LIN {X 0,Y 489.995,Z 461.229,A -85,B 0,C 180,E1 -6434.645,E2 -6434.645} C_VEL
LIN {X 0,Y 490.457,Z 449.449,A -85,B 0,C 180,E1 -6435.4,E2 -6435.4} C_VEL
LIN {X 0,Y 490.746,Z 438.449,A -85,B 0,C 180,E1 -6435.942,E2 -6435.942} C_VEL
LIN {X 0,Y 490.984,Z 425.122,A -85,B 0,C 180,E1 -6436.413,E2 -6436.413} C_VEL
LIN {X 0,Y 491.19,Z 412.427,A -85,B 0,C 180,E1 -6436.693,E2 -6436.693} C_VEL
LIN {X 0,Y 491.72,Z 322.911,A -85,B 0,C 180,E1 -6438.028,E2 -6438.028} C_VEL
LIN {X 0,Y 489.317,Z 310.007,A -85,B 0,C 180,E1 -6438.311,E2 -6438.311} C_VEL
LIN {X 0,Y 489.405,Z 294.541,A -85,B 0,C 180,E1 -6441.085,E2 -6441.085} C_VEL
LIN {X 0,Y 488.713,Z 289.612,A -85,B 0,C 180,E1 -6442.025,E2 -6442.025} C_VEL
LIN {X 0,Y 488.689,Z 289.61,A -85,B 0,C 180,E1 -6445.048,E2 -6445.048} C_VEL
LIN {X 0,Y 488.664,Z 289.617,A -85,B 0,C 180,E1 -6448.042,E2 -6448.042} C_VEL
LIN {X 0,Y 488.689,Z 289.612,A -85,B 0,C 180,E1 -6450.727,E2 -6450.727} C_VEL
LIN {X 0,Y 488.721,Z 289.607,A -85,B 0,C 180,E1 -6453.526,E2 -6453.526} C_VEL
LIN {X 0,Y 488.645,Z 289.623,A -85,B 0,C 180,E1 -6456.252,E2 -6456.252} C_VEL
LIN {X 0,Y 488.696,Z 289.609,A -85,B 0,C 180,E1 -6459.173,E2 -6459.173} C_VEL
LIN {X 0,Y 488.682,Z 289.616,A -85,B 0,C 180,E1 -6462.421,E2 -6462.421} C_VEL
LIN {X 0,Y 488.708,Z 289.609,A -85,B 0,C 180,E1 -6464.998,E2 -6464.998} C_VEL
LIN {X 0,Y 488.754,Z 289.604,A -85,B 0,C 180,E1 -6468.386,E2 -6468.386} C_VEL
LIN {X 0,Y 488.763,Z 289.598,A -85,B 0,C 180,E1 -6471.733,E2 -6471.733} C_VEL
LIN {X 0,Y 488.8,Z 289.595,A -85,B 0,C 180,E1 -6474.224,E2 -6474.224} C_VEL
LIN {X 0,Y 488.909,Z 289.58,A -85,B 0,C 180,E1 -6477.528,E2 -6477.528} C_VEL
LIN {X 0,Y 488.909,Z 289.576,A -85,B 0,C 180,E1 -6480,E2 -6480} C_VEL
LIN {X 0,Y 488.911,Z 289.582,A -85,B 0,C 180,E1 -6482.472,E2 -6482.472} C_VEL
LIN {X 0,Y 488.818,Z 289.591,A -85,B 0,C 180,E1 -6485.776,E2 -6485.776} C_VEL
LIN {X 0,Y 488.772,Z 289.594,A -85,B 0,C 180,E1 -6488.267,E2 -6488.267} C_VEL
LIN {X 0,Y 488.781,Z 289.594,A -85,B 0,C 180,E1 -6491.613,E2 -6491.613} C_VEL
LIN {X 0,Y 488.718,Z 289.61,A -85,B 0,C 180,E1 -6495.002,E2 -6495.002} C_VEL
LIN {X 0,Y 488.704,Z 289.604,A -85,B 0,C 180,E1 -6498.444,E2 -6498.444} C_VEL
LIN {X 0,Y 488.695,Z 289.608,A -85,B 0,C 180,E1 -6501.071,E2 -6501.071} C_VEL
LIN {X 0,Y 488.671,Z 289.608,A -85,B 0,C 180,E1 -6503.747,E2 -6503.747} C_VEL
LIN {X 0,Y 488.753,Z 289.601,A -85,B 0,C 180,E1 -6506.948,E2 -6506.948} C_VEL
LIN {X 0,Y 488.676,Z 289.608,A -85,B 0,C 180,E1 -6510.368,E2 -6510.368} C_VEL
LIN {X 0,Y 488.695,Z 289.615,A -85,B 0,C 180,E1 -6513.488,E2 -6513.488} C_VEL
LIN {X 0,Y 488.661,Z 289.611,A -85,B 0,C 180,E1 -6516.361,E2 -6516.361} C_VEL
LIN {X 0,Y 488.724,Z 289.606,A -85,B 0,C 180,E1 -6519.252,E2 -6519.252} C_VEL
LIN {X 0,Y 488.7,Z 289.608,A -85,B 0,C 180,E1 -6522.525,E2 -6522.525} C_VEL
LIN {X 0,Y 488.681,Z 289.613,A -85,B 0,C 180,E1 -6525.203,E2 -6525.203} C_VEL
LIN {X 0,Y 488.705,Z 289.613,A -85,B 0,C 180,E1 -6527.483,E2 -6527.483} C_VEL
LIN {X 0,Y 488.743,Z 289.61,A -85,B 0,C 180,E1 -6529.684,E2 -6529.684} C_VEL
LIN {X 0,Y 488.662,Z 289.611,A -85,B 0,C 180,E1 -6532.846,E2 -6532.846} C_VEL
LIN {X 0,Y 488.715,Z 289.612,A -85,B 0,C 180,E1 -6535.892,E2 -6535.892} C_VEL
LIN {X 0,Y 488.679,Z 289.613,A -85,B 0,C 180,E1 -6538.825,E2 -6538.825} C_VEL
LIN {X 0,Y 488.731,Z 289.61,A -85,B 0,C 180,E1 -6541.676,E2 -6541.676} C_VEL
LIN {X 0,Y 488.783,Z 289.603,A -85,B 0,C 180,E1 -6544.698,E2 -6544.698} C_VEL
LIN {X 0,Y 490.547,Z 299.643,A -85,B 0,C 180,E1 -6546.48,E2 -6546.48} C_VEL
LIN {X 0,Y 490.042,Z 317.608,A -85,B 0,C 180,E1 -6549.433,E2 -6549.433} C_VEL
LIN {X 0,Y 489.438,Z 336.212,A -85,B 0,C 180,E1 -6552.454,E2 -6552.454} C_VEL
LIN {X 0,Y 489.242,Z 344.16,A -85,B 0,C 180,E1 -6553.726,E2 -6553.726} C_VEL
LIN {X 0,Y 491.661,Z 361.485,A -85,B 0,C 180,E1 -6554.069,E2 -6554.069} C_VEL
LIN {X 0,Y 491.029,Z 452.97,A -85,B 0,C 180,E1 -6555.445,E2 -6555.445} C_VEL
LIN {X 0,Y 490.645,Z 466.878,A -85,B 0,C 180,E1 -6555.831,E2 -6555.831} C_VEL
LIN {X 0,Y 490.312,Z 479.869,A -85,B 0,C 180,E1 -6556.376,E2 -6556.376} C_VEL
LIN {X 0,Y 489.937,Z 492.098,A -85,B 0,C 180,E1 -6557.079,E2 -6557.079} C_VEL
LIN {X 0,Y 489.544,Z 503.076,A -85,B 0,C 180,E1 -6557.884,E2 -6557.884} C_VEL
LIN {X 0,Y 489.135,Z 513.353,A -85,B 0,C 180,E1 -6558.819,E2 -6558.819} C_VEL
LIN {X 0,Y 488.745,Z 522.589,A -85,B 0,C 180,E1 -6559.858,E2 -6559.858} C_VEL
LIN {X 0,Y 488.43,Z 531.587,A -85,B 0,C 180,E1 -6561.105,E2 -6561.105} C_VEL
LIN {X 0,Y 488.205,Z 538.835,A -85,B 0,C 180,E1 -6562.351,E2 -6562.351} C_VEL
LIN {X 0,Y 488.047,Z 544.326,A -85,B 0,C 180,E1 -6563.525,E2 -6563.525} C_VEL
LIN {X 0,Y 488.017,Z 548.484,A -85,B 0,C 180,E1 -6564.632,E2 -6564.632} C_VEL
LIN {X 0,Y 487.928,Z 552.119,A -85,B 0,C 180,E1 -6565.873,E2 -6565.873} C_VEL
LIN {X 0,Y 487.964,Z 553.997,A -85,B 0,C 180,E1 -6566.7,E2 -6566.7} C_VEL
LIN {X 0,Y 487.89,Z 556.408,A -85,B 0,C 180,E1 -6568.352,E2 -6568.352} C_VEL
LIN {X 0,Y 487.822,Z 557.242,A -85,B 0,C 180,E1 -6570.003,E2 -6570.003} C_VEL
LIN {X 0,Y 487.891,Z 556.422,A -85,B 0,C 180,E1 -6571.653,E2 -6571.653} C_VEL
LIN {X 0,Y 487.909,Z 555.425,A -85,B 0,C 180,E1 -6572.479,E2 -6572.479} C_VEL
LIN {X 0,Y 487.965,Z 554.025,A -85,B 0,C 180,E1 -6573.305,E2 -6573.305} C_VEL
LIN {X 0,Y 487.921,Z 551.075,A -85,B 0,C 180,E1 -6574.546,E2 -6574.546} C_VEL
LIN {X 0,Y 488.023,Z 547.084,A -85,B 0,C 180,E1 -6575.788,E2 -6575.788} C_VEL
LIN {X 0,Y 488.183,Z 540.94,A -85,B 0,C 180,E1 -6577.239,E2 -6577.239} C_VEL
LIN {X 0,Y 488.355,Z 534.227,A -85,B 0,C 180,E1 -6578.485,E2 -6578.485} C_VEL
LIN {X 0,Y 488.648,Z 525.9,A -85,B 0,C 180,E1 -6579.731,E2 -6579.731} C_VEL
LIN {X 0,Y 488.977,Z 517.349,A -85,B 0,C 180,E1 -6580.771,E2 -6580.771} C_VEL
LIN {X 0,Y 489.449,Z 506.791,A -85,B 0,C 180,E1 -6581.809,E2 -6581.809} C_VEL
LIN {X 0,Y 489.741,Z 496.622,A -85,B 0,C 180,E1 -6582.622,E2 -6582.622} C_VEL
LIN {X 0,Y 490.159,Z 484.852,A -85,B 0,C 180,E1 -6583.37,E2 -6583.37} C_VEL
LIN {X 0,Y 490.521,Z 472.979,A -85,B 0,C 180,E1 -6583.94,E2 -6583.94} C_VEL
LIN {X 0,Y 490.9,Z 459.284,A -85,B 0,C 180,E1 -6584.405,E2 -6584.405} C_VEL
LIN {X 0,Y 491.115,Z 446.975,A -85,B 0,C 180,E1 -6584.664,E2 -6584.664} C_VEL
LIN {X 0,Y 491.634,Z 360.174,A -85,B 0,C 180,E1 -6585.951,E2 -6585.951} C_VEL
LIN {X 0,Y 489.29,Z 344.503,A -85,B 0,C 180,E1 -6586.268,E2 -6586.268} C_VEL
LIN {X 0,Y 489.908,Z 324.958,A -85,B 0,C 180,E1 -6589.485,E2 -6589.485} C_VEL
LIN {X 0,Y 490.513,Z 307.991,A -85,B 0,C 180,E1 -6592.316,E2 -6592.316} C_VEL
LIN {X 0,Y 490.718,Z 300.156,A -85,B 0,C 180,E1 -6593.643,E2 -6593.643} C_VEL
LIN {X 0,Y 488.808,Z 289.599,A -85,B 0,C 180,E1 -6595.582,E2 -6595.582} C_VEL
LIN {X 0,Y 488.733,Z 289.605,A -85,B 0,C 180,E1 -6598.695,E2 -6598.695} C_VEL
LIN {X 0,Y 488.696,Z 289.608,A -85,B 0,C 180,E1 -6601.18,E2 -6601.18} C_VEL
LIN {X 0,Y 488.734,Z 289.609,A -85,B 0,C 180,E1 -6604.113,E2 -6604.113} C_VEL
LIN {X 0,Y 488.681,Z 289.607,A -85,B 0,C 180,E1 -6607.159,E2 -6607.159} C_VEL
LIN {X 0,Y 488.72,Z 289.611,A -85,B 0,C 180,E1 -6610.345,E2 -6610.345} C_VEL
LIN {X 0,Y 488.684,Z 289.607,A -85,B 0,C 180,E1 -6613.655,E2 -6613.655} C_VEL
LIN {X 0,Y 488.683,Z 289.615,A -85,B 0,C 180,E1 -6616.345,E2 -6616.345} C_VEL
LIN {X 0,Y 488.732,Z 289.601,A -85,B 0,C 180,E1 -6619.676,E2 -6619.676} C_VEL
LIN {X 0,Y 488.679,Z 289.613,A -85,B 0,C 180,E1 -6622.841,E2 -6622.841} C_VEL
LIN {X 0,Y 488.729,Z 289.602,A -85,B 0,C 180,E1 -6625.887,E2 -6625.887} C_VEL
LIN {X 0,Y 488.69,Z 289.614,A -85,B 0,C 180,E1 -6628.82,E2 -6628.82} C_VEL
LIN {X 0,Y 488.74,Z 289.6,A -85,B 0,C 180,E1 -6631.671,E2 -6631.671} C_VEL
LIN {X 0,Y 488.741,Z 289.603,A -85,B 0,C 180,E1 -6634.444,E2 -6634.444} C_VEL
LIN {X 0,Y 488.716,Z 289.609,A -85,B 0,C 180,E1 -6637.153,E2 -6637.153} C_VEL
LIN {X 0,Y 488.716,Z 289.603,A -85,B 0,C 180,E1 -6639.81,E2 -6639.81} C_VEL
LIN {X 0,Y 488.719,Z 289.604,A -85,B 0,C 180,E1 -6642.423,E2 -6642.423} C_VEL
LIN {X 0,Y 488.752,Z 289.606,A -85,B 0,C 180,E1 -6644.999,E2 -6644.999} C_VEL
LIN {X 0,Y 488.796,Z 289.593,A -85,B 0,C 180,E1 -6648.387,E2 -6648.387} C_VEL
LIN {X 0,Y 488.806,Z 289.595,A -85,B 0,C 180,E1 -6651.733,E2 -6651.733} C_VEL
LIN {X 0,Y 488.835,Z 289.588,A -85,B 0,C 180,E1 -6654.224,E2 -6654.224} C_VEL
LIN {X 0,Y 488.947,Z 289.582,A -85,B 0,C 180,E1 -6657.529,E2 -6657.529} C_VEL
LIN {X 0,Y 488.953,Z 289.576,A -85,B 0,C 180,E1 -6660,E2 -6660} C_VEL
LIN {X 0,Y 488.946,Z 289.574,A -85,B 0,C 180,E1 -6662.471,E2 -6662.471} C_VEL
LIN {X 0,Y 488.825,Z 289.596,A -85,B 0,C 180,E1 -6665.776,E2 -6665.776} C_VEL
LIN {X 0,Y 488.774,Z 289.597,A -85,B 0,C 180,E1 -6668.267,E2 -6668.267} C_VEL
LIN {X 0,Y 488.794,Z 289.6,A -85,B 0,C 180,E1 -6671.613,E2 -6671.613} C_VEL
LIN {X 0,Y 488.747,Z 289.599,A -85,B 0,C 180,E1 -6675.001,E2 -6675.001} C_VEL
LIN {X 0,Y 488.736,Z 289.602,A -85,B 0,C 180,E1 -6678.443,E2 -6678.443} C_VEL
LIN {X 0,Y 488.698,Z 289.605,A -85,B 0,C 180,E1 -6681.071,E2 -6681.071} C_VEL
LIN {X 0,Y 488.661,Z 289.614,A -85,B 0,C 180,E1 -6683.747,E2 -6683.747} C_VEL
LIN {X 0,Y 488.689,Z 289.607,A -85,B 0,C 180,E1 -6686.922,E2 -6686.922} C_VEL
LIN {X 0,Y 488.711,Z 289.613,A -85,B 0,C 180,E1 -6690.22,E2 -6690.22} C_VEL
LIN {X 0,Y 488.704,Z 289.605,A -85,B 0,C 180,E1 -6693.48,E2 -6693.48} C_VEL
LIN {X 0,Y 488.643,Z 289.622,A -85,B 0,C 180,E1 -6696.349,E2 -6696.349} C_VEL
LIN {X 0,Y 488.667,Z 289.609,A -85,B 0,C 180,E1 -6699.258,E2 -6699.258} C_VEL
LIN {X 0,Y 488.645,Z 289.621,A -85,B 0,C 180,E1 -6702.531,E2 -6702.531} C_VEL
LIN {X 0,Y 488.694,Z 289.607,A -85,B 0,C 180,E1 -6705.197,E2 -6705.197} C_VEL
LIN {X 0,Y 488.642,Z 289.62,A -85,B 0,C 180,E1 -6708.578,E2 -6708.578} C_VEL
LIN {X 0,Y 488.641,Z 289.612,A -85,B 0,C 180,E1 -6711.796,E2 -6711.796} C_VEL
LIN {X 0,Y 488.634,Z 289.618,A -85,B 0,C 180,E1 -6715.068,E2 -6715.068} C_VEL
LIN {X 0,Y 488.684,Z 289.607,A -85,B 0,C 180,E1 -6718.05,E2 -6718.05} C_VEL
LIN {X 0,Y 488.663,Z 289.613,A -85,B 0,C 180,E1 -6721.32,E2 -6721.32} C_VEL
LIN {X 0,Y 488.648,Z 289.612,A -85,B 0,C 180,E1 -6724.325,E2 -6724.325} C_VEL
LIN {X 0,Y 488.009,Z 289.7,A -85,B 0,C 180,E1 -6725.014,E2 -6725.014} C_VEL
LIN {X 0,Y 485.179,Z 290.049,A -85,B 0,C 180,E1 -6726.132,E2 -6726.132} C_VEL
LIN {X 0,Y 482.768,Z 290.352,A -85,B 0,C 180,E1 -6727.033,E2 -6727.033} C_VEL
LIN {X 0,Y 481.727,Z 290.475,A -85,B 0,C 180,E1 -6727.728,E2 -6727.728} C_VEL
LIN {X 0,Y 481.639,Z 290.485,A -85,B 0,C 180,E1 -6727.964,E2 -6727.964} C_VEL
LIN {X 0,Y 481.699,Z 290.477,A -85,B 0,C 180,E1 -6730.391,E2 -6730.391} C_VEL
LIN {X 0,Y 481.662,Z 290.488,A -85,B 0,C 180,E1 -6733.031,E2 -6733.031} C_VEL
LIN {X 0,Y 481.681,Z 290.483,A -85,B 0,C 180,E1 -6735.637,E2 -6735.637} C_VEL
LIN {X 0,Y 481.755,Z 290.47,A -85,B 0,C 180,E1 -6738.213,E2 -6738.213} C_VEL
LIN {X 0,Y 481.721,Z 290.481,A -85,B 0,C 180,E1 -6741.609,E2 -6741.609} C_VEL
LIN {X 0,Y 481.778,Z 290.468,A -85,B 0,C 180,E1 -6744.137,E2 -6744.137} C_VEL
LIN {X 0,Y 481.91,Z 290.459,A -85,B 0,C 180,E1 -6747.49,E2 -6747.49} C_VEL
LIN {X 0,Y 481.913,Z 290.454,A -85,B 0,C 180,E1 -6749.997,E2 -6749.997} C_VEL
LIN {X 0,Y 481.911,Z 290.451,A -85,B 0,C 180,E1 -6752.505,E2 -6752.505} C_VEL
LIN {X 0,Y 481.777,Z 290.476,A -85,B 0,C 180,E1 -6755.858,E2 -6755.858} C_VEL
LIN {X 0,Y 481.734,Z 290.478,A -85,B 0,C 180,E1 -6758.385,E2 -6758.385} C_VEL
LIN {X 0,Y 481.772,Z 290.586,A -85,B 0,C 180,E1 -6761.461,E2 -6761.461} C_VEL
LIN {X 0,Y 482.681,Z 297.868,A -85,B 0,C 180,E1 -6762.997,E2 -6762.997} C_VEL
LIN {X 0,Y 482.362,Z 310.521,A -85,B 0,C 180,E1 -6765.551,E2 -6765.551} C_VEL
LIN {X 0,Y 484.964,Z 324.373,A -85,B 0,C 180,E1 -6765.864,E2 -6765.864} C_VEL
LIN {X 0,Y 484.213,Z 417.892,A -85,B 0,C 180,E1 -6767.292,E2 -6767.292} C_VEL
LIN {X 0,Y 484.01,Z 431.131,A -85,B 0,C 180,E1 -6767.668,E2 -6767.668} C_VEL
LIN {X 0,Y 483.711,Z 443.779,A -85,B 0,C 180,E1 -6768.199,E2 -6768.199} C_VEL
LIN {X 0,Y 483.25,Z 455.563,A -85,B 0,C 180,E1 -6768.869,E2 -6768.869} C_VEL
LIN {X 0,Y 482.785,Z 467.826,A -85,B 0,C 180,E1 -6769.778,E2 -6769.778} C_VEL
LIN {X 0,Y 482.382,Z 477.231,A -85,B 0,C 180,E1 -6770.65,E2 -6770.65} C_VEL
LIN {X 0,Y 482.013,Z 485.672,A -85,B 0,C 180,E1 -6771.598,E2 -6771.598} C_VEL
LIN {X 0,Y 481.717,Z 494.021,A -85,B 0,C 180,E1 -6772.74,E2 -6772.74} C_VEL
LIN {X 0,Y 481.397,Z 502.142,A -85,B 0,C 180,E1 -6774.123,E2 -6774.123} C_VEL
LIN {X 0,Y 481.155,Z 508.6,A -85,B 0,C 180,E1 -6775.519,E2 -6775.519} C_VEL
LIN {X 0,Y 480.993,Z 513.665,A -85,B 0,C 180,E1 -6776.963,E2 -6776.963} C_VEL
LIN {X 0,Y 480.913,Z 516.158,A -85,B 0,C 180,E1 -6777.876,E2 -6777.876} C_VEL
LIN {X 0,Y 480.803,Z 518.209,A -85,B 0,C 180,E1 -6778.835,E2 -6778.835} C_VEL
LIN {X 0,Y 480.751,Z 520.365,A -85,B 0,C 180,E1 -6780.4,E2 -6780.4} C_VEL
LIN {X 0,Y 480.727,Z 521.162,A -85,B 0,C 180,E1 -6782.012,E2 -6782.012} C_VEL
LIN {X 0,Y 480.727,Z 520.513,A -85,B 0,C 180,E1 -6783.559,E2 -6783.559} C_VEL
LIN {X 0,Y 480.813,Z 518.588,A -85,B 0,C 180,E1 -6785.06,E2 -6785.06} C_VEL
LIN {X 0,Y 480.947,Z 515.464,A -85,B 0,C 180,E1 -6786.514,E2 -6786.514} C_VEL
LIN {X 0,Y 481.061,Z 511.182,A -85,B 0,C 180,E1 -6787.916,E2 -6787.916} C_VEL
LIN {X 0,Y 481.256,Z 505.608,A -85,B 0,C 180,E1 -6789.287,E2 -6789.287} C_VEL
LIN {X 0,Y 481.54,Z 498.625,A -85,B 0,C 180,E1 -6790.63,E2 -6790.63} C_VEL
LIN {X 0,Y 481.869,Z 490.094,A -85,B 0,C 180,E1 -6791.941,E2 -6791.941} C_VEL
LIN {X 0,Y 482.312,Z 480.839,A -85,B 0,C 180,E1 -6793.074,E2 -6793.074} C_VEL
LIN {X 0,Y 482.732,Z 471.215,A -85,B 0,C 180,E1 -6794.034,E2 -6794.034} C_VEL
LIN {X 0,Y 483.112,Z 460.087,A -85,B 0,C 180,E1 -6794.932,E2 -6794.932} C_VEL
LIN {X 0,Y 483.562,Z 448.087,A -85,B 0,C 180,E1 -6795.683,E2 -6795.683} C_VEL
LIN {X 0,Y 483.945,Z 435.708,A -85,B 0,C 180,E1 -6796.265,E2 -6796.265} C_VEL
LIN {X 0,Y 484.208,Z 423.12,A -85,B 0,C 180,E1 -6796.684,E2 -6796.684} C_VEL
LIN {X 0,Y 484.385,Z 408.413,A -85,B 0,C 180,E1 -6796.97,E2 -6796.97} C_VEL
LIN {X 0,Y 484.909,Z 323.537,A -85,B 0,C 180,E1 -6798.257,E2 -6798.257} C_VEL
LIN {X 0,Y 482.363,Z 310.099,A -85,B 0,C 180,E1 -6798.58,E2 -6798.58} C_VEL
LIN {X 0,Y 482.459,Z 295.54,A -85,B 0,C 180,E1 -6801.216,E2 -6801.216} C_VEL
LIN {X 0,Y 481.662,Z 290.491,A -85,B 0,C 180,E1 -6802.206,E2 -6802.206} C_VEL
LIN {X 0,Y 481.653,Z 290.487,A -85,B 0,C 180,E1 -6805.315,E2 -6805.315} C_VEL
LIN {X 0,Y 481.606,Z 290.497,A -85,B 0,C 180,E1 -6808.309,E2 -6808.309} C_VEL
LIN {X 0,Y 481.661,Z 290.484,A -85,B 0,C 180,E1 -6811.216,E2 -6811.216} C_VEL
LIN {X 0,Y 481.66,Z 290.491,A -85,B 0,C 180,E1 -6814.04,E2 -6814.04} C_VEL
LIN {X 0,Y 481.626,Z 290.494,A -85,B 0,C 180,E1 -6816.809,E2 -6816.809} C_VEL
LIN {X 0,Y 481.645,Z 290.487,A -85,B 0,C 180,E1 -6819.5,E2 -6819.5} C_VEL
LIN {X 0,Y 481.655,Z 290.488,A -85,B 0,C 180,E1 -6822.156,E2 -6822.156} C_VEL
LIN {X 0,Y 481.689,Z 290.486,A -85,B 0,C 180,E1 -6824.774,E2 -6824.774} C_VEL
LIN {X 0,Y 481.699,Z 290.481,A -85,B 0,C 180,E1 -6828.214,E2 -6828.214} C_VEL
LIN {X 0,Y 481.709,Z 290.477,A -85,B 0,C 180,E1 -6831.611,E2 -6831.611} C_VEL
LIN {X 0,Y 481.759,Z 290.471,A -85,B 0,C 180,E1 -6834.139,E2 -6834.139} C_VEL
LIN {X 0,Y 481.878,Z 290.456,A -85,B 0,C 180,E1 -6837.492,E2 -6837.492} C_VEL
LIN {X 0,Y 481.881,Z 290.451,A -85,B 0,C 180,E1 -6840,E2 -6840} C_VEL
LIN {X 0,Y 481.88,Z 290.458,A -85,B 0,C 180,E1 -6842.508,E2 -6842.508} C_VEL
LIN {X 0,Y 481.776,Z 290.468,A -85,B 0,C 180,E1 -6845.861,E2 -6845.861} C_VEL
LIN {X 0,Y 481.718,Z 290.473,A -85,B 0,C 180,E1 -6848.389,E2 -6848.389} C_VEL
LIN {X 0,Y 481.745,Z 290.469,A -85,B 0,C 180,E1 -6851.785,E2 -6851.785} C_VEL
LIN {X 0,Y 481.696,Z 290.482,A -85,B 0,C 180,E1 -6855.226,E2 -6855.226} C_VEL
LIN {X 0,Y 481.663,Z 290.484,A -85,B 0,C 180,E1 -6858.724,E2 -6858.724} C_VEL
LIN {X 0,Y 481.632,Z 290.491,A -85,B 0,C 180,E1 -6861.395,E2 -6861.395} C_VEL
LIN {X 0,Y 481.652,Z 290.479,A -85,B 0,C 180,E1 -6864.115,E2 -6864.115} C_VEL
LIN {X 0,Y 481.707,Z 290.481,A -85,B 0,C 180,E1 -6867.143,E2 -6867.143} C_VEL
LIN {X 0,Y 481.645,Z 290.488,A -85,B 0,C 180,E1 -6869.744,E2 -6869.744} C_VEL
LIN {X 0,Y 481.633,Z 290.485,A -85,B 0,C 180,E1 -6872.677,E2 -6872.677} C_VEL
LIN {X 0,Y 481.612,Z 290.496,A -85,B 0,C 180,E1 -6875.712,E2 -6875.712} C_VEL
LIN {X 0,Y 481.681,Z 290.48,A -85,B 0,C 180,E1 -6878.858,E2 -6878.858} C_VEL
LIN {X 0,Y 481.642,Z 290.49,A -85,B 0,C 180,E1 -6882.161,E2 -6882.161} C_VEL
LIN {X 0,Y 481.628,Z 290.49,A -85,B 0,C 180,E1 -6884.461,E2 -6884.461} C_VEL
LIN {X 0,Y 481.659,Z 290.486,A -85,B 0,C 180,E1 -6886.85,E2 -6886.85} C_VEL
LIN {X 0,Y 481.687,Z 290.486,A -85,B 0,C 180,E1 -6890.067,E2 -6890.067} C_VEL
LIN {X 0,Y 481.61,Z 290.492,A -85,B 0,C 180,E1 -6893.379,E2 -6893.379} C_VEL
LIN {X 0,Y 481.689,Z 290.486,A -85,B 0,C 180,E1 -6896.334,E2 -6896.334} C_VEL
LIN {X 0,Y 481.641,Z 290.492,A -85,B 0,C 180,E1 -6899.42,E2 -6899.42} C_VEL
LIN {X 0,Y 481.688,Z 290.487,A -85,B 0,C 180,E1 -6902.172,E2 -6902.172} C_VEL
LIN {X 0,Y 481.753,Z 290.562,A -85,B 0,C 180,E1 -6904.541,E2 -6904.541} C_VEL
LIN {X 0,Y 483.56,Z 300.365,A -85,B 0,C 180,E1 -6906.296,E2 -6906.296} C_VEL
LIN {X 0,Y 483.123,Z 315.977,A -85,B 0,C 180,E1 -6908.902,E2 -6908.902} C_VEL
LIN {X 0,Y 482.538,Z 334.623,A -85,B 0,C 180,E1 -6911.975,E2 -6911.975} C_VEL
LIN {X 0,Y 482.239,Z 343.798,A -85,B 0,C 180,E1 -6913.477,E2 -6913.477} C_VEL
LIN {X 0,Y 484.842,Z 361.274,A -85,B 0,C 180,E1 -6913.839,E2 -6913.839} C_VEL
LIN {X 0,Y 484.163,Z 452.637,A -85,B 0,C 180,E1 -6915.234,E2 -6915.234} C_VEL
LIN {X 0,Y 483.819,Z 465.8,A -85,B 0,C 180,E1 -6915.6,E2 -6915.6} C_VEL
LIN {X 0,Y 483.429,Z 478.495,A -85,B 0,C 180,E1 -6916.125,E2 -6916.125} C_VEL
LIN {X 0,Y 483.051,Z 490.113,A -85,B 0,C 180,E1 -6916.778,E2 -6916.778} C_VEL
LIN {X 0,Y 482.584,Z 501.481,A -85,B 0,C 180,E1 -6917.599,E2 -6917.599} C_VEL
LIN {X 0,Y 482.169,Z 512.004,A -85,B 0,C 180,E1 -6918.549,E2 -6918.549} C_VEL
LIN {X 0,Y 481.796,Z 520.608,A -85,B 0,C 180,E1 -6919.497,E2 -6919.497} C_VEL
LIN {X 0,Y 481.469,Z 528.548,A -85,B 0,C 180,E1 -6920.552,E2 -6920.552} C_VEL
LIN {X 0,Y 481.222,Z 536.307,A -85,B 0,C 180,E1 -6921.817,E2 -6921.817} C_VEL
LIN {X 0,Y 481.005,Z 543.454,A -85,B 0,C 180,E1 -6923.291,E2 -6923.291} C_VEL
LIN {X 0,Y 480.93,Z 548.214,A -85,B 0,C 180,E1 -6924.553,E2 -6924.553} C_VEL
LIN {X 0,Y 480.828,Z 551.85,A -85,B 0,C 180,E1 -6925.812,E2 -6925.812} C_VEL
LIN {X 0,Y 480.887,Z 553.731,A -85,B 0,C 180,E1 -6926.652,E2 -6926.652} C_VEL
LIN {X 0,Y 480.82,Z 556.144,A -85,B 0,C 180,E1 -6928.328,E2 -6928.328} C_VEL
LIN {X 0,Y 480.745,Z 556.978,A -85,B 0,C 180,E1 -6930.003,E2 -6930.003} C_VEL
LIN {X 0,Y 480.821,Z 556.159,A -85,B 0,C 180,E1 -6931.678,E2 -6931.678} C_VEL
LIN {X 0,Y 480.889,Z 553.759,A -85,B 0,C 180,E1 -6933.354,E2 -6933.354} C_VEL
LIN {X 0,Y 480.839,Z 550.807,A -85,B 0,C 180,E1 -6934.613,E2 -6934.613} C_VEL
LIN {X 0,Y 480.927,Z 546.812,A -85,B 0,C 180,E1 -6935.874,E2 -6935.874} C_VEL
LIN {X 0,Y 481.108,Z 540.661,A -85,B 0,C 180,E1 -6937.346,E2 -6937.346} C_VEL
LIN {X 0,Y 481.308,Z 533.944,A -85,B 0,C 180,E1 -6938.61,E2 -6938.61} C_VEL
LIN {X 0,Y 481.593,Z 525.609,A -85,B 0,C 180,E1 -6939.875,E2 -6939.875} C_VEL
LIN {X 0,Y 481.97,Z 517.049,A -85,B 0,C 180,E1 -6940.929,E2 -6940.929} C_VEL
LIN {X 0,Y 482.463,Z 506.504,A -85,B 0,C 180,E1 -6941.98,E2 -6941.98} C_VEL
LIN {X 0,Y 482.852,Z 495.228,A -85,B 0,C 180,E1 -6942.885,E2 -6942.885} C_VEL
LIN {X 0,Y 483.223,Z 484.511,A -85,B 0,C 180,E1 -6943.565,E2 -6943.565} C_VEL
LIN {X 0,Y 483.626,Z 472.607,A -85,B 0,C 180,E1 -6944.143,E2 -6944.143} C_VEL
LIN {X 0,Y 484.02,Z 458.871,A -85,B 0,C 180,E1 -6944.615,E2 -6944.615} C_VEL
LIN {X 0,Y 484.245,Z 446.434,A -85,B 0,C 180,E1 -6944.876,E2 -6944.876} C_VEL
LIN {X 0,Y 484.779,Z 360.639,A -85,B 0,C 180,E1 -6946.169,E2 -6946.169} C_VEL
LIN {X 0,Y 482.269,Z 344.236,A -85,B 0,C 180,E1 -6946.511,E2 -6946.511} C_VEL
LIN {X 0,Y 482.921,Z 325.998,A -85,B 0,C 180,E1 -6949.557,E2 -6949.557} C_VEL
LIN {X 0,Y 483.583,Z 309.05,A -85,B 0,C 180,E1 -6952.428,E2 -6952.428} C_VEL
LIN {X 0,Y 483.753,Z 301.335,A -85,B 0,C 180,E1 -6953.756,E2 -6953.756} C_VEL
LIN {X 0,Y 481.766,Z 290.477,A -85,B 0,C 180,E1 -6955.775,E2 -6955.775} C_VEL
LIN {X 0,Y 481.68,Z 290.483,A -85,B 0,C 180,E1 -6958.903,E2 -6958.903} C_VEL
LIN {X 0,Y 481.661,Z 290.49,A -85,B 0,C 180,E1 -6962.189,E2 -6962.189} C_VEL
LIN {X 0,Y 481.691,Z 290.48,A -85,B 0,C 180,E1 -6964.682,E2 -6964.682} C_VEL
LIN {X 0,Y 481.656,Z 290.488,A -85,B 0,C 180,E1 -6968.007,E2 -6968.007} C_VEL
LIN {X 0,Y 481.658,Z 290.483,A -85,B 0,C 180,E1 -6971.042,E2 -6971.042} C_VEL
LIN {X 0,Y 481.655,Z 290.491,A -85,B 0,C 180,E1 -6974.458,E2 -6974.458} C_VEL
LIN {X 0,Y 481.647,Z 290.485,A -85,B 0,C 180,E1 -6977.839,E2 -6977.839} C_VEL
LIN {X 0,Y 481.678,Z 290.487,A -85,B 0,C 180,E1 -6980.651,E2 -6980.651} C_VEL
LIN {X 0,Y 481.627,Z 290.486,A -85,B 0,C 180,E1 -6983.376,E2 -6983.376} C_VEL
LIN {X 0,Y 481.707,Z 290.48,A -85,B 0,C 180,E1 -6986.33,E2 -6986.33} C_VEL
LIN {X 0,Y 481.648,Z 290.484,A -85,B 0,C 180,E1 -6989.417,E2 -6989.417} C_VEL
LIN {X 0,Y 481.695,Z 290.479,A -85,B 0,C 180,E1 -6992.168,E2 -6992.168} C_VEL
LIN {X 0,Y 481.712,Z 290.483,A -85,B 0,C 180,E1 -6994.969,E2 -6994.969} C_VEL
LIN {X 0,Y 481.641,Z 290.485,A -85,B 0,C 180,E1 -6997.704,E2 -6997.704} C_VEL
LIN {X 0,Y 481.696,Z 290.479,A -85,B 0,C 180,E1 -7000.393,E2 -7000.393} C_VEL
LIN {X 0,Y 481.678,Z 290.488,A -85,B 0,C 180,E1 -7003.033,E2 -7003.033} C_VEL
LIN {X 0,Y 481.679,Z 290.482,A -85,B 0,C 180,E1 -7005.638,E2 -7005.638} C_VEL
LIN {X 0,Y 481.741,Z 290.472,A -85,B 0,C 180,E1 -7008.215,E2 -7008.215} C_VEL
LIN {X 0,Y 481.752,Z 290.475,A -85,B 0,C 180,E1 -7011.612,E2 -7011.612} C_VEL
LIN {X 0,Y 481.796,Z 290.465,A -85,B 0,C 180,E1 -7014.139,E2 -7014.139} C_VEL
LIN {X 0,Y 481.915,Z 290.458,A -85,B 0,C 180,E1 -7017.492,E2 -7017.492} C_VEL
LIN {X 0,Y 481.924,Z 290.451,A -85,B 0,C 180,E1 -7020,E2 -7020} C_VEL
LIN {X 0,Y 481.913,Z 290.45,A -85,B 0,C 180,E1 -7022.508,E2 -7022.508} C_VEL
LIN {X 0,Y 481.784,Z 290.472,A -85,B 0,C 180,E1 -7025.861,E2 -7025.861} C_VEL
LIN {X 0,Y 481.729,Z 290.474,A -85,B 0,C 180,E1 -7028.389,E2 -7028.389} C_VEL
LIN {X 0,Y 481.74,Z 290.481,A -85,B 0,C 180,E1 -7031.785,E2 -7031.785} C_VEL
LIN {X 0,Y 481.73,Z 290.474,A -85,B 0,C 180,E1 -7035.225,E2 -7035.225} C_VEL
LIN {X 0,Y 481.698,Z 290.477,A -85,B 0,C 180,E1 -7038.722,E2 -7038.722} C_VEL
LIN {X 0,Y 481.635,Z 290.486,A -85,B 0,C 180,E1 -7041.395,E2 -7041.395} C_VEL
LIN {X 0,Y 481.64,Z 290.493,A -85,B 0,C 180,E1 -7044.115,E2 -7044.115} C_VEL
LIN {X 0,Y 481.644,Z 290.484,A -85,B 0,C 180,E1 -7047.117,E2 -7047.117} C_VEL
LIN {X 0,Y 481.659,Z 290.485,A -85,B 0,C 180,E1 -7049.743,E2 -7049.743} C_VEL
LIN {X 0,Y 481.647,Z 290.487,A -85,B 0,C 180,E1 -7052.676,E2 -7052.676} C_VEL
LIN {X 0,Y 481.644,Z 290.484,A -85,B 0,C 180,E1 -7055.202,E2 -7055.202} C_VEL
LIN {X 0,Y 481.622,Z 290.49,A -85,B 0,C 180,E1 -7058.003,E2 -7058.003} C_VEL
LIN {X 0,Y 481.602,Z 290.491,A -85,B 0,C 180,E1 -7061.048,E2 -7061.048} C_VEL
LIN {X 0,Y 481.649,Z 290.491,A -85,B 0,C 180,E1 -7064.459,E2 -7064.459} C_VEL
LIN {X 0,Y 481.608,Z 290.489,A -85,B 0,C 180,E1 -7067.835,E2 -7067.835} C_VEL
LIN {X 0,Y 481.628,Z 290.495,A -85,B 0,C 180,E1 -7070.659,E2 -7070.659} C_VEL
LIN {X 0,Y 481.585,Z 290.492,A -85,B 0,C 180,E1 -7073.383,E2 -7073.383} C_VEL
LIN {X 0,Y 481.608,Z 290.491,A -85,B 0,C 180,E1 -7076.321,E2 -7076.321} C_VEL
LIN {X 0,Y 481.613,Z 290.49,A -85,B 0,C 180,E1 -7079.426,E2 -7079.426} C_VEL
LIN {X 0,Y 481.645,Z 290.484,A -85,B 0,C 180,E1 -7082.164,E2 -7082.164} C_VEL
LIN {X 0,Y 481.669,Z 290.489,A -85,B 0,C 180,E1 -7084.966,E2 -7084.966} C_VEL
LIN {X 0,Y 481.639,Z 290.485,A -85,B 0,C 180,E1 -7087.964,E2 -7087.964} C_VEL
LIN {X 0,Y 480.973,Z 290.571,A -85,B 0,C 180,E1 -7088.662,E2 -7088.662} C_VEL
LIN {X 0,Y 478.15,Z 290.925,A -85,B 0,C 180,E1 -7089.796,E2 -7089.796} C_VEL
LIN {X 0,Y 475.763,Z 291.224,A -85,B 0,C 180,E1 -7090.711,E2 -7090.711} C_VEL
LIN {X 0,Y 474.733,Z 291.351,A -85,B 0,C 180,E1 -7091.416,E2 -7091.416} C_VEL
LIN {X 0,Y 474.646,Z 291.358,A -85,B 0,C 180,E1 -7091.655,E2 -7091.655} C_VEL
LIN {X 0,Y 474.702,Z 291.349,A -85,B 0,C 180,E1 -7094.543,E2 -7094.543} C_VEL
LIN {X 0,Y 474.709,Z 291.349,A -85,B 0,C 180,E1 -7098.036,E2 -7098.036} C_VEL
LIN {X 0,Y 474.67,Z 291.361,A -85,B 0,C 180,E1 -7101.483,E2 -7101.483} C_VEL
LIN {X 0,Y 474.741,Z 291.345,A -85,B 0,C 180,E1 -7104.05,E2 -7104.05} C_VEL
LIN {X 0,Y 474.875,Z 291.334,A -85,B 0,C 180,E1 -7107.453,E2 -7107.453} C_VEL
LIN {X 0,Y 474.882,Z 291.33,A -85,B 0,C 180,E1 -7109.997,E2 -7109.997} C_VEL
LIN {X 0,Y 474.876,Z 291.327,A -85,B 0,C 180,E1 -7112.542,E2 -7112.542} C_VEL
LIN {X 0,Y 474.74,Z 291.353,A -85,B 0,C 180,E1 -7115.945,E2 -7115.945} C_VEL
LIN {X 0,Y 474.706,Z 291.353,A -85,B 0,C 180,E1 -7118.511,E2 -7118.511} C_VEL
LIN {X 0,Y 474.74,Z 291.515,A -85,B 0,C 180,E1 -7121.308,E2 -7121.308} C_VEL
LIN {X 0,Y 475.707,Z 298.563,A -85,B 0,C 180,E1 -7122.819,E2 -7122.819} C_VEL
LIN {X 0,Y 475.415,Z 310.966,A -85,B 0,C 180,E1 -7125.318,E2 -7125.318} C_VEL
LIN {X 0,Y 478.175,Z 325.002,A -85,B 0,C 180,E1 -7125.637,E2 -7125.637} C_VEL
LIN {X 0,Y 477.366,Z 418.042,A -85,B 0,C 180,E1 -7127.078,E2 -7127.078} C_VEL
LIN {X 0,Y 477.138,Z 431.363,A -85,B 0,C 180,E1 -7127.46,E2 -7127.46} C_VEL
LIN {X 0,Y 476.819,Z 443.449,A -85,B 0,C 180,E1 -7127.971,E2 -7127.971} C_VEL
LIN {X 0,Y 476.422,Z 454.585,A -85,B 0,C 180,E1 -7128.598,E2 -7128.598} C_VEL
LIN {X 0,Y 475.942,Z 466.187,A -85,B 0,C 180,E1 -7129.445,E2 -7129.445} C_VEL
LIN {X 0,Y 475.429,Z 476.995,A -85,B 0,C 180,E1 -7130.436,E2 -7130.436} C_VEL
LIN {X 0,Y 475.001,Z 486.835,A -85,B 0,C 180,E1 -7131.563,E2 -7131.563} C_VEL
LIN {X 0,Y 474.64,Z 495.552,A -85,B 0,C 180,E1 -7132.807,E2 -7132.807} C_VEL
LIN {X 0,Y 474.365,Z 502.554,A -85,B 0,C 180,E1 -7134.039,E2 -7134.039} C_VEL
LIN {X 0,Y 474.091,Z 508.982,A -85,B 0,C 180,E1 -7135.456,E2 -7135.456} C_VEL
LIN {X 0,Y 473.937,Z 513.597,A -85,B 0,C 180,E1 -7136.777,E2 -7136.777} C_VEL
LIN {X 0,Y 473.764,Z 517.572,A -85,B 0,C 180,E1 -7138.335,E2 -7138.335} C_VEL
LIN {X 0,Y 473.687,Z 519.354,A -85,B 0,C 180,E1 -7139.31,E2 -7139.31} C_VEL
LIN {X 0,Y 473.644,Z 520.852,A -85,B 0,C 180,E1 -7140.614,E2 -7140.614} C_VEL
LIN {X 0,Y 473.632,Z 521.392,A -85,B 0,C 180,E1 -7142.283,E2 -7142.283} C_VEL
LIN {X 0,Y 473.647,Z 520.572,A -85,B 0,C 180,E1 -7143.805,E2 -7143.805} C_VEL
LIN {X 0,Y 473.753,Z 518.455,A -85,B 0,C 180,E1 -7145.343,E2 -7145.343} C_VEL
LIN {X 0,Y 473.895,Z 515.204,A -85,B 0,C 180,E1 -7146.79,E2 -7146.79} C_VEL
LIN {X 0,Y 474.04,Z 510.705,A -85,B 0,C 180,E1 -7148.208,E2 -7148.208} C_VEL
LIN {X 0,Y 474.276,Z 504.93,A -85,B 0,C 180,E1 -7149.596,E2 -7149.596} C_VEL
LIN {X 0,Y 474.585,Z 497.771,A -85,B 0,C 180,E1 -7150.953,E2 -7150.953} C_VEL
LIN {X 0,Y 474.838,Z 490.808,A -85,B 0,C 180,E1 -7152.024,E2 -7152.024} C_VEL
LIN {X 0,Y 475.284,Z 482.083,A -85,B 0,C 180,E1 -7153.13,E2 -7153.13} C_VEL
LIN {X 0,Y 475.734,Z 472.553,A -85,B 0,C 180,E1 -7154.113,E2 -7154.113} C_VEL
LIN {X 0,Y 476.136,Z 462.653,A -85,B 0,C 180,E1 -7154.949,E2 -7154.949} C_VEL
LIN {X 0,Y 476.622,Z 451.147,A -85,B 0,C 180,E1 -7155.723,E2 -7155.723} C_VEL
LIN {X 0,Y 476.994,Z 440.396,A -85,B 0,C 180,E1 -7156.285,E2 -7156.285} C_VEL
LIN {X 0,Y 477.265,Z 427.908,A -85,B 0,C 180,E1 -7156.768,E2 -7156.768} C_VEL
LIN {X 0,Y 477.476,Z 414.661,A -85,B 0,C 180,E1 -7157.093,E2 -7157.093} C_VEL
LIN {X 0,Y 478.148,Z 324.496,A -85,B 0,C 180,E1 -7158.486,E2 -7158.486} C_VEL
LIN {X 0,Y 475.438,Z 310.369,A -85,B 0,C 180,E1 -7158.829,E2 -7158.829} C_VEL
LIN {X 0,Y 475.515,Z 296.512,A -85,B 0,C 180,E1 -7161.359,E2 -7161.359} C_VEL
LIN {X 0,Y 474.611,Z 291.369,A -85,B 0,C 180,E1 -7162.35,E2 -7162.35} C_VEL
LIN {X 0,Y 474.594,Z 291.369,A -85,B 0,C 180,E1 -7165.756,E2 -7165.756} C_VEL
LIN {X 0,Y 474.56,Z 291.372,A -85,B 0,C 180,E1 -7168.779,E2 -7168.779} C_VEL
LIN {X 0,Y 474.605,Z 291.365,A -85,B 0,C 180,E1 -7171.715,E2 -7171.715} C_VEL
LIN {X 0,Y 474.623,Z 291.369,A -85,B 0,C 180,E1 -7174.575,E2 -7174.575} C_VEL
LIN {X 0,Y 474.552,Z 291.372,A -85,B 0,C 180,E1 -7177.353,E2 -7177.353} C_VEL
LIN {X 0,Y 474.604,Z 291.368,A -85,B 0,C 180,E1 -7180.087,E2 -7180.087} C_VEL
LIN {X 0,Y 474.598,Z 291.368,A -85,B 0,C 180,E1 -7182.772,E2 -7182.772} C_VEL
LIN {X 0,Y 474.594,Z 291.364,A -85,B 0,C 180,E1 -7185.419,E2 -7185.419} C_VEL
LIN {X 0,Y 474.652,Z 291.358,A -85,B 0,C 180,E1 -7188.036,E2 -7188.036} C_VEL
LIN {X 0,Y 474.674,Z 291.353,A -85,B 0,C 180,E1 -7191.485,E2 -7191.485} C_VEL
LIN {X 0,Y 474.721,Z 291.348,A -85,B 0,C 180,E1 -7194.052,E2 -7194.052} C_VEL
LIN {X 0,Y 474.845,Z 291.333,A -85,B 0,C 180,E1 -7197.455,E2 -7197.455} C_VEL
LIN {X 0,Y 474.824,Z 291.339,A -85,B 0,C 180,E1 -7200.848,E2 -7200.848} C_VEL
LIN {X 0,Y 474.847,Z 291.335,A -85,B 0,C 180,E1 -7202.545,E2 -7202.545} C_VEL
LIN {X 0,Y 474.736,Z 291.345,A -85,B 0,C 180,E1 -7205.948,E2 -7205.948} C_VEL
LIN {X 0,Y 474.683,Z 291.35,A -85,B 0,C 180,E1 -7208.514,E2 -7208.514} C_VEL
LIN {X 0,Y 474.688,Z 291.347,A -85,B 0,C 180,E1 -7211.963,E2 -7211.963} C_VEL
LIN {X 0,Y 474.652,Z 291.353,A -85,B 0,C 180,E1 -7215.779,E2 -7215.779} C_VEL
LIN {X 0,Y 474.616,Z 291.365,A -85,B 0,C 180,E1 -7219.012,E2 -7219.012} C_VEL
LIN {X 0,Y 474.599,Z 291.364,A -85,B 0,C 180,E1 -7221.728,E2 -7221.728} C_VEL
LIN {X 0,Y 474.631,Z 291.354,A -85,B 0,C 180,E1 -7224.494,E2 -7224.494} C_VEL
LIN {X 0,Y 474.654,Z 291.36,A -85,B 0,C 180,E1 -7227.342,E2 -7227.342} C_VEL
LIN {X 0,Y 474.568,Z 291.367,A -85,B 0,C 180,E1 -7230.815,E2 -7230.815} C_VEL
LIN {X 0,Y 474.598,Z 291.364,A -85,B 0,C 180,E1 -7233.988,E2 -7233.988} C_VEL
LIN {X 0,Y 474.549,Z 291.37,A -85,B 0,C 180,E1 -7236.905,E2 -7236.905} C_VEL
LIN {X 0,Y 474.637,Z 291.367,A -85,B 0,C 180,E1 -7239.658,E2 -7239.658} C_VEL
LIN {X 0,Y 474.619,Z 291.363,A -85,B 0,C 180,E1 -7242.934,E2 -7242.934} C_VEL
LIN {X 0,Y 474.588,Z 291.372,A -85,B 0,C 180,E1 -7245.9,E2 -7245.9} C_VEL
LIN {X 0,Y 474.62,Z 291.363,A -85,B 0,C 180,E1 -7249.042,E2 -7249.042} C_VEL
LIN {X 0,Y 474.596,Z 291.371,A -85,B 0,C 180,E1 -7251.707,E2 -7251.707} C_VEL
LIN {X 0,Y 474.609,Z 291.364,A -85,B 0,C 180,E1 -7254.731,E2 -7254.731} C_VEL
LIN {X 0,Y 474.619,Z 291.371,A -85,B 0,C 180,E1 -7257.792,E2 -7257.792} C_VEL
LIN {X 0,Y 474.616,Z 291.365,A -85,B 0,C 180,E1 -7260.887,E2 -7260.887} C_VEL
LIN {X 0,Y 474.659,Z 291.362,A -85,B 0,C 180,E1 -7263.633,E2 -7263.633} C_VEL
LIN {X 0,Y 474.684,Z 291.404,A -85,B 0,C 180,E1 -7264.334,E2 -7264.334} C_VEL
LIN {X 0,Y 476.641,Z 301.947,A -85,B 0,C 180,E1 -7266.256,E2 -7266.256} C_VEL
LIN {X 0,Y 476.14,Z 318.372,A -85,B 0,C 180,E1 -7269.034,E2 -7269.034} C_VEL
LIN {X 0,Y 475.416,Z 338.324,A -85,B 0,C 180,E1 -7272.363,E2 -7272.363} C_VEL
LIN {X 0,Y 475.245,Z 343.51,A -85,B 0,C 180,E1 -7273.223,E2 -7273.223} C_VEL
LIN {X 0,Y 478.04,Z 362.231,A -85,B 0,C 180,E1 -7273.618,E2 -7273.618} C_VEL
LIN {X 0,Y 477.289,Z 452.353,A -85,B 0,C 180,E1 -7275.017,E2 -7275.017} C_VEL
LIN {X 0,Y 476.919,Z 466.265,A -85,B 0,C 180,E1 -7275.414,E2 -7275.414} C_VEL
LIN {X 0,Y 476.501,Z 478.191,A -85,B 0,C 180,E1 -7275.919,E2 -7275.919} C_VEL
LIN {X 0,Y 476.104,Z 489.498,A -85,B 0,C 180,E1 -7276.56,E2 -7276.56} C_VEL
LIN {X 0,Y 475.666,Z 500.496,A -85,B 0,C 180,E1 -7277.358,E2 -7277.358} C_VEL
LIN {X 0,Y 475.191,Z 511.716,A -85,B 0,C 180,E1 -7278.378,E2 -7278.378} C_VEL
LIN {X 0,Y 474.76,Z 520.323,A -85,B 0,C 180,E1 -7279.34,E2 -7279.34} C_VEL
LIN {X 0,Y 474.441,Z 528.268,A -85,B 0,C 180,E1 -7280.41,E2 -7280.41} C_VEL
LIN {X 0,Y 474.159,Z 536.03,A -85,B 0,C 180,E1 -7281.694,E2 -7281.694} C_VEL
LIN {X 0,Y 473.923,Z 543.181,A -85,B 0,C 180,E1 -7283.19,E2 -7283.19} C_VEL
LIN {X 0,Y 473.844,Z 547.944,A -85,B 0,C 180,E1 -7284.471,E2 -7284.471} C_VEL
LIN {X 0,Y 473.734,Z 551.582,A -85,B 0,C 180,E1 -7285.749,E2 -7285.749} C_VEL
LIN {X 0,Y 473.794,Z 553.464,A -85,B 0,C 180,E1 -7286.601,E2 -7286.601} C_VEL
LIN {X 0,Y 473.74,Z 554.872,A -85,B 0,C 180,E1 -7287.452,E2 -7287.452} C_VEL
LIN {X 0,Y 473.723,Z 555.879,A -85,B 0,C 180,E1 -7288.303,E2 -7288.303} C_VEL
LIN {X 0,Y 473.688,Z 556.495,A -85,B 0,C 180,E1 -7289.153,E2 -7289.153} C_VEL
LIN {X 0,Y 473.672,Z 556.715,A -85,B 0,C 180,E1 -7290.003,E2 -7290.003} C_VEL
LIN {X 0,Y 473.689,Z 556.5,A -85,B 0,C 180,E1 -7290.853,E2 -7290.853} C_VEL
LIN {X 0,Y 473.724,Z 555.893,A -85,B 0,C 180,E1 -7291.703,E2 -7291.703} C_VEL
LIN {X 0,Y 473.742,Z 554.895,A -85,B 0,C 180,E1 -7292.553,E2 -7292.553} C_VEL
LIN {X 0,Y 473.796,Z 553.491,A -85,B 0,C 180,E1 -7293.404,E2 -7293.404} C_VEL
LIN {X 0,Y 473.763,Z 550.537,A -85,B 0,C 180,E1 -7294.682,E2 -7294.682} C_VEL
LIN {X 0,Y 473.834,Z 546.538,A -85,B 0,C 180,E1 -7295.962,E2 -7295.962} C_VEL
LIN {X 0,Y 474.016,Z 540.381,A -85,B 0,C 180,E1 -7297.456,E2 -7297.456} C_VEL
LIN {X 0,Y 474.254,Z 533.659,A -85,B 0,C 180,E1 -7298.739,E2 -7298.739} C_VEL
LIN {X 0,Y 474.555,Z 525.318,A -85,B 0,C 180,E1 -7300.023,E2 -7300.023} C_VEL
LIN {X 0,Y 474.955,Z 516.748,A -85,B 0,C 180,E1 -7301.093,E2 -7301.093} C_VEL
LIN {X 0,Y 475.461,Z 506.44,A -85,B 0,C 180,E1 -7302.137,E2 -7302.137} C_VEL
LIN {X 0,Y 475.857,Z 495.981,A -85,B 0,C 180,E1 -7302.996,E2 -7302.996} C_VEL
LIN {X 0,Y 476.305,Z 484.17,A -85,B 0,C 180,E1 -7303.766,E2 -7303.766} C_VEL
LIN {X 0,Y 476.784,Z 470.936,A -85,B 0,C 180,E1 -7304.405,E2 -7304.405} C_VEL
LIN {X 0,Y 477.189,Z 457.531,A -85,B 0,C 180,E1 -7304.856,E2 -7304.856} C_VEL
LIN {X 0,Y 477.429,Z 442.335,A -85,B 0,C 180,E1 -7305.148,E2 -7305.148} C_VEL
LIN {X 0,Y 477.859,Z 361.041,A -85,B 0,C 180,E1 -7306.396,E2 -7306.396} C_VEL
LIN {X 0,Y 475.29,Z 343.961,A -85,B 0,C 180,E1 -7306.761,E2 -7306.761} C_VEL
LIN {X 0,Y 475.962,Z 325.739,A -85,B 0,C 180,E1 -7309.855,E2 -7309.855} C_VEL
LIN {X 0,Y 476.64,Z 310.093,A -85,B 0,C 180,E1 -7312.544,E2 -7312.544} C_VEL
LIN {X 0,Y 476.734,Z 302.153,A -85,B 0,C 180,E1 -7313.935,E2 -7313.935} C_VEL
LIN {X 0,Y 474.692,Z 291.359,A -85,B 0,C 180,E1 -7315.989,E2 -7315.989} C_VEL
LIN {X 0,Y 474.648,Z 291.363,A -85,B 0,C 180,E1 -7318.283,E2 -7318.283} C_VEL
LIN {X 0,Y 474.603,Z 291.364,A -85,B 0,C 180,E1 -7321.218,E2 -7321.218} C_VEL
LIN {X 0,Y 474.636,Z 291.365,A -85,B 0,C 180,E1 -7324.241,E2 -7324.241} C_VEL
LIN {X 0,Y 474.592,Z 291.362,A -85,B 0,C 180,E1 -7327.384,E2 -7327.384} C_VEL
LIN {X 0,Y 474.619,Z 291.363,A -85,B 0,C 180,E1 -7330.658,E2 -7330.658} C_VEL
LIN {X 0,Y 474.596,Z 291.362,A -85,B 0,C 180,E1 -7333.48,E2 -7333.48} C_VEL
LIN {X 0,Y 474.595,Z 291.37,A -85,B 0,C 180,E1 -7336.52,E2 -7336.52} C_VEL
LIN {X 0,Y 474.616,Z 291.36,A -85,B 0,C 180,E1 -7339.342,E2 -7339.342} C_VEL
LIN {X 0,Y 474.608,Z 291.36,A -85,B 0,C 180,E1 -7341.704,E2 -7341.704} C_VEL
LIN {X 0,Y 474.625,Z 291.366,A -85,B 0,C 180,E1 -7344.726,E2 -7344.726} C_VEL
LIN {X 0,Y 474.633,Z 291.357,A -85,B 0,C 180,E1 -7347.787,E2 -7347.787} C_VEL
LIN {X 0,Y 474.62,Z 291.367,A -85,B 0,C 180,E1 -7350.884,E2 -7350.884} C_VEL
LIN {X 0,Y 474.654,Z 291.355,A -85,B 0,C 180,E1 -7353.628,E2 -7353.628} C_VEL
LIN {X 0,Y 474.63,Z 291.362,A -85,B 0,C 180,E1 -7356.641,E2 -7356.641} C_VEL
LIN {X 0,Y 474.646,Z 291.356,A -85,B 0,C 180,E1 -7360.089,E2 -7360.089} C_VEL
LIN {X 0,Y 474.638,Z 291.361,A -85,B 0,C 180,E1 -7362.774,E2 -7362.774} C_VEL
LIN {X 0,Y 474.638,Z 291.361,A -85,B 0,C 180,E1 -7365.421,E2 -7365.421} C_VEL
LIN {X 0,Y 474.695,Z 291.35,A -85,B 0,C 180,E1 -7368.037,E2 -7368.037} C_VEL
LIN {X 0,Y 474.718,Z 291.353,A -85,B 0,C 180,E1 -7371.486,E2 -7371.486} C_VEL
LIN {X 0,Y 474.759,Z 291.342,A -85,B 0,C 180,E1 -7374.052,E2 -7374.052} C_VEL
LIN {X 0,Y 474.881,Z 291.335,A -85,B 0,C 180,E1 -7377.455,E2 -7377.455} C_VEL
LIN {X 0,Y 474.895,Z 291.327,A -85,B 0,C 180,E1 -7380,E2 -7380} C_VEL
LIN {X 0,Y 474.88,Z 291.326,A -85,B 0,C 180,E1 -7382.545,E2 -7382.545} C_VEL
LIN {X 0,Y 474.745,Z 291.348,A -85,B 0,C 180,E1 -7385.948,E2 -7385.948} C_VEL
LIN {X 0,Y 474.701,Z 291.349,A -85,B 0,C 180,E1 -7388.514,E2 -7388.514} C_VEL
LIN {X 0,Y 474.694,Z 291.356,A -85,B 0,C 180,E1 -7391.963,E2 -7391.963} C_VEL
LIN {X 0,Y 474.689,Z 291.354,A -85,B 0,C 180,E1 -7395.456,E2 -7395.456} C_VEL
LIN {X 0,Y 474.652,Z 291.355,A -85,B 0,C 180,E1 -7399.011,E2 -7399.011} C_VEL
LIN {X 0,Y 474.578,Z 291.369,A -85,B 0,C 180,E1 -7401.73,E2 -7401.73} C_VEL
LIN {X 0,Y 474.618,Z 291.362,A -85,B 0,C 180,E1 -7404.495,E2 -7404.495} C_VEL
LIN {X 0,Y 474.59,Z 291.363,A -85,B 0,C 180,E1 -7407.327,E2 -7407.327} C_VEL
LIN {X 0,Y 474.591,Z 291.371,A -85,B 0,C 180,E1 -7410.231,E2 -7410.231} C_VEL
LIN {X 0,Y 474.61,Z 291.36,A -85,B 0,C 180,E1 -7413.223,E2 -7413.223} C_VEL
LIN {X 0,Y 474.565,Z 291.375,A -85,B 0,C 180,E1 -7416.326,E2 -7416.326} C_VEL
LIN {X 0,Y 474.596,Z 291.362,A -85,B 0,C 180,E1 -7419.551,E2 -7419.551} C_VEL
LIN {X 0,Y 474.563,Z 291.369,A -85,B 0,C 180,E1 -7422.94,E2 -7422.94} C_VEL
LIN {X 0,Y 474.566,Z 291.366,A -85,B 0,C 180,E1 -7425.89,E2 -7425.89} C_VEL
LIN {X 0,Y 474.58,Z 291.367,A -85,B 0,C 180,E1 -7429.048,E2 -7429.048} C_VEL
LIN {X 0,Y 474.581,Z 291.364,A -85,B 0,C 180,E1 -7431.709,E2 -7431.709} C_VEL
LIN {X 0,Y 474.544,Z 291.376,A -85,B 0,C 180,E1 -7434.718,E2 -7434.718} C_VEL
LIN {X 0,Y 474.609,Z 291.36,A -85,B 0,C 180,E1 -7437.785,E2 -7437.785} C_VEL
LIN {X 0,Y 474.578,Z 291.373,A -85,B 0,C 180,E1 -7440.895,E2 -7440.895} C_VEL
LIN {X 0,Y 474.574,Z 291.366,A -85,B 0,C 180,E1 -7443.622,E2 -7443.622} C_VEL
LIN {X 0,Y 474.639,Z 291.359,A -85,B 0,C 180,E1 -7446.641,E2 -7446.641} C_VEL
LIN {X 0,Y 474.652,Z 291.355,A -85,B 0,C 180,E1 -7450.088,E2 -7450.088} C_VEL
LIN {X 0,Y 474.646,Z 291.358,A -85,B 0,C 180,E1 -7451.655,E2 -7451.655} C_VEL
LIN {X 0,Y 473.973,Z 291.44,A -85,B 0,C 180,E1 -7452.364,E2 -7452.364} C_VEL
LIN {X 0,Y 471.125,Z 291.8,A -85,B 0,C 180,E1 -7453.515,E2 -7453.515} C_VEL
LIN {X 0,Y 468.719,Z 292.104,A -85,B 0,C 180,E1 -7454.444,E2 -7454.444} C_VEL
LIN {X 0,Y 467.681,Z 292.231,A -85,B 0,C 180,E1 -7455.161,E2 -7455.161} C_VEL
LIN {X 0,Y 467.594,Z 292.239,A -85,B 0,C 180,E1 -7455.403,E2 -7455.403} C_VEL
LIN {X 0,Y 467.661,Z 292.228,A -85,B 0,C 180,E1 -7457.853,E2 -7457.853} C_VEL
LIN {X 0,Y 467.639,Z 292.237,A -85,B 0,C 180,E1 -7461.354,E2 -7461.354} C_VEL
LIN {X 0,Y 467.706,Z 292.223,A -85,B 0,C 180,E1 -7463.96,E2 -7463.96} C_VEL
LIN {X 0,Y 467.815,Z 292.213,A -85,B 0,C 180,E1 -7467.414,E2 -7467.414} C_VEL
LIN {X 0,Y 467.852,Z 292.206,A -85,B 0,C 180,E1 -7469.997,E2 -7469.997} C_VEL
LIN {X 0,Y 467.816,Z 292.206,A -85,B 0,C 180,E1 -7472.58,E2 -7472.58} C_VEL
